(* IEC 61131-3 sources: Codesys/60-let-oktyabrya/src, 26 files *)

(* ---- E_PumpType.st ---- *)
(* ============================================================ *)
(* E_PumpType — тип преобразователя частоты ELHART             *)
(* ============================================================ *)
(* === ИЗМЕНЕНО === MINI удалён (в проектах его не было — была   *)
(* ошибка типа). Теперь два типа: PUMP (EMD-PUMP) и VL           *)
(* (EMD-VL/VH, векторный). Обработка обоих — в FB_Pump.          *)
(*                                                              *)
(* Тип каждого ПЧ задаётся в массиве GVL.ePumpType[1..cPumpCount] *)
(* (RETAIN). Автоопределение PUMP/VL по сигнатурному регистру —   *)
(* см. комментарий в PRG_Pumps (пока задаётся вручную).          *)
(* ============================================================ *)
TYPE E_PumpType :
(
    PUMP := 0,   // EMD-PUMP (F-коды, задание частоты в Гц ×100 → 0x2001)
    VL   := 1    // EMD-VL (P-группы, задание в % → 0x1000, статус 0x3000)
);
END_TYPE

(* ---- GVL.st ---- *)
(* ============================================================ *)
(* GVL — Глобальные переменные проекта "60 Лет Октября"         *)
(* (на основе ДДЮТ / Fontan_V1 / Саки Пруд)                     *)
(*                                                              *)
(* ШИНА Modbus RTU / RS-485:                                   *)
(*   COM1 (Modbus_COM), 9600/8/N/1:                            *)
(*     Адрес 1  — МВ110-16Д   (16 дискретных входов DI1..DI12) *)
(*     Адрес 2  — МУ110-16Р   (16 дискретных выходов DO1..DO4  *)
(*                используются, остальные свободны)             *)
(*   COM2 (Modbus_COM_2):                                       *)
(*     Адрес 41 — ELHART EMD-PUMP 1 (насос-шоу, индекс 1)      *)
(*     Адрес 42 — ELHART EMD-PUMP 2 (насос-шоу, индекс 2)      *)
(*     Адрес 43 — ELHART EMD-PUMP 3 (насос-шоу, индекс 3, НОВЫЙ)*)
(*     === 60ЛО:ВАЖНО === Устройство EMD_PUMP_3 нужно добавить  *)
(*     в дереве Modbus проекта (по аналогии с EMD_PUMP_1/2) —    *)
(*     без него PRG_Pumps.st (блок 4а) не скомпилируется.        *)
(*   ПЧ COM2 — насосы-шоу (не фильтрационные), просто            *)
(*   информационные, ни на что в логике не влияют.               *)
(* ============================================================ *)

(* ============================================================ *)
(* КОНСТАНТЫ СИСТЕМЫ                                            *)
(* ============================================================ *)
VAR_GLOBAL CONSTANT
    cPumpCount   : INT  := 3;        // === 60ЛО:ИЗМЕНЕНО === было 2 (ДДЮТ), теперь 3 насоса ПЧ (ПЧ1/ПЧ2/ПЧ3)
    cDI_Count    : INT  := 16;       // дискретных входов МВ110
    cDO_Count    : INT  := 16;       // дискретных выходов МУ110
    cMaxFreq     : REAL := 50.0;     // максимальная частота, Гц
    cMinFreq     : REAL := 0.0;      // минимальная частота, Гц
    cMinTime     : REAL := 0.1;      // мин. время разгона/торможения, с
    cMaxTime     : REAL := 6000.0;   // макс. время разгона/торможения, с
    cMaxCurrent  : REAL := 999.9;    // потолок номинального тока, А
    cMaxVoltage  : REAL := 500.0;    // потолок номинального напряжения, В
    cMaxOverheat : INT  := 150;      // потолок уровня перегрева, °C
    cMinOverheat : INT  := 40;       // минимум уровня перегрева, °C
END_VAR

(* ============================================================ *)
(* RETAIN-переменные (хранятся при отключении питания)         *)
(* ============================================================ *)
VAR_GLOBAL RETAIN
    (* Тип каждого ПЧ. Все три насоса — EMD-PUMP.                *)
    (* ВНИМАНИЕ: изменение требует Reset cold контроллера.      *)
    ePumpType : ARRAY[1..cPumpCount] OF E_PumpType :=
        [E_PumpType.PUMP, E_PumpType.PUMP, E_PumpType.PUMP];   // === 60ЛО:ИЗМЕНЕНО === добавлен 3-й элемент

    (* === ЖУРНАЛ ПЧ — БЕЗ ИЗМЕНЕНИЙ АРХИТЕКТУРЫ === *)
    (* Та же схема сдвига, что у журнала фонтана (см. подробный комментарий  *)
    (* в GVL_Fountain.st) — позиция 1 всегда самая свежая запись, при новой  *)
    (* записи всё сдвигается на 1 вниз, самая старая (позиция 30) выпадает.  *)
    (* Размер: 30 записей, длина ячейки 65.                                  *)
    (* ⚠️ С полными названиями возможна обрезка длинных строк — если         *)
    (* увидишь обрыв текста, увеличь до 80-90).                              *)
    aPumpLog       : ARRAY[1..30] OF WSTRING(65);
    iPumpLogCount  : INT;   // сколько записей реально заполнено (0..30)

    (* Флаг "задержка ошибки 0x02C0 уже записана в ПЧ" — RETAIN *)
    xErrDelayWritten : ARRAY[1..cPumpCount] OF BOOL := [cPumpCount(FALSE)];

    (* Флаг "параметр дисплея Fout (регистр 0) уже записан" — RETAIN *)
    xDispParamWritten : ARRAY[1..cPumpCount] OF BOOL := [cPumpCount(FALSE)];
END_VAR

(* ============================================================ *)
(* ГЛОБАЛЬНЫЕ ПЕРЕМЕННЫЕ                                        *)
(* ============================================================ *)
VAR_GLOBAL

    (* ========================================================= *)
    (* БЛОК 1: СОСТОЯНИЕ СИСТЕМЫ                                 *)
    (* ========================================================= *)
    xSystemState     : BOOL := TRUE;
    sSystemStateText : WSTRING(20);
    iErrors          : INT  := 0;
    iWorkCount       : INT  := 0;
    iStopCount       : INT  := 0;
    xAnyAlarm        : BOOL := FALSE;
    iErrorsPumps     : INT  := 0;
    iErrorsModules   : INT  := 0;
    iErrorsFountain  : INT  := 0;

    (* ========================================================= *)
    (* БЛОК 2: НАВИГАЦИЯ И ИНТЕРФЕЙС HMI                         *)
    (* ========================================================= *)
    xMenuOpen      : BOOL := TRUE;
    iCurrentScreen : INT  := 1;
    iSelPump       : INT  := 1;

    (* ========================================================= *)
    (* БЛОК 3: РЕЖИМ ОТЛАДКИ RS-485                              *)
    (* ========================================================= *)
    xDebugModeAll      : BOOL := FALSE;
    xDebugModeAll_Prev : BOOL := FALSE;

    xDebugModePump      : ARRAY[1..cPumpCount] OF BOOL := [cPumpCount(FALSE)];
    xDebugModePump_Prev : ARRAY[1..cPumpCount] OF BOOL := [cPumpCount(FALSE)];

    xApplyParamsAll  : BOOL := FALSE;
    xApplyParamsPump : ARRAY[1..cPumpCount] OF BOOL := [cPumpCount(FALSE)];

    (* ========================================================= *)
    (* ТРИГГЕРЫ ЧТЕНИЯ/ЗАПИСИ (конфигуратор-стиль)               *)
    (* ========================================================= *)
    xReadAllPump  : ARRAY[1..cPumpCount] OF BOOL := [cPumpCount(FALSE)];
    xReadAllAsk   : BOOL := FALSE;

    xWriteAllPump : ARRAY[1..cPumpCount] OF BOOL := [cPumpCount(FALSE)];
    xWriteAllAsk  : BOOL := FALSE;
    xWriteAllConfirm : BOOL := FALSE;

    xWr_AccTime      : ARRAY[1..cPumpCount] OF BOOL := [cPumpCount(FALSE)]; // 0x006B
    xWr_DecTime      : ARRAY[1..cPumpCount] OF BOOL := [cPumpCount(FALSE)]; // 0x006C
    xWr_MaxFreq      : ARRAY[1..cPumpCount] OF BOOL := [cPumpCount(FALSE)]; // 0x0069
    xWr_MinFreq      : ARRAY[1..cPumpCount] OF BOOL := [cPumpCount(FALSE)]; // 0x006A
    xWr_MotorCurrent : ARRAY[1..cPumpCount] OF BOOL := [cPumpCount(FALSE)]; // 0x00D2
    xWr_MotorVoltage : ARRAY[1..cPumpCount] OF BOOL := [cPumpCount(FALSE)]; // 0x00D1
    xWr_OverCurLevel : ARRAY[1..cPumpCount] OF BOOL := [cPumpCount(FALSE)]; // 0x01A7
    xWr_OverCurTime  : ARRAY[1..cPumpCount] OF BOOL := [cPumpCount(FALSE)]; // 0x01A8
    xWr_OverVoltProt : ARRAY[1..cPumpCount] OF BOOL := [cPumpCount(FALSE)]; // 0x019B
    xWr_Overheat     : ARRAY[1..cPumpCount] OF BOOL := [cPumpCount(FALSE)]; // 0x0325
    xWr_OverCurAcc   : ARRAY[1..cPumpCount] OF BOOL := [cPumpCount(FALSE)]; // 0x0199

    xWr_UnlockF800   : ARRAY[1..cPumpCount] OF BOOL := [cPumpCount(FALSE)]; // 0x0320
    xWr_Sources      : ARRAY[1..cPumpCount] OF BOOL := [cPumpCount(FALSE)]; // 0x0065/0x0066

    xWritePending    : ARRAY[1..cPumpCount] OF BOOL := [cPumpCount(FALSE)];
    xWaitStopForWrite : ARRAY[1..cPumpCount] OF BOOL := [cPumpCount(FALSE)];

    (* === 60ЛО:УДАЛИТЬ ===                                       *)
    (* Раньше использовался для запроса физической остановки      *)
    (* фильтр.насоса через лампы DO6/DO8 перед записью параметров. *)
    (* Не читается нигде физически, оставлен только для истории.  *)
    xReqStopFiltrForWrite : ARRAY[1..cPumpCount] OF BOOL := [cPumpCount(FALSE)];

    xFactoryResetAll  : BOOL := FALSE;
    xFactoryResetPump : ARRAY[1..cPumpCount] OF BOOL := [cPumpCount(FALSE)];

    wCmdSourceWrite  : ARRAY[1..cPumpCount] OF WORD := [cPumpCount(WORD#1)];
    wFreqSourceWrite : ARRAY[1..cPumpCount] OF WORD := [cPumpCount(WORD#3)];

    (* ========================================================= *)
    (* БЛОК 4: МВ110-16Д — ДИСКРЕТНЫЕ ВХОДЫ                      *)
    (* ========================================================= *)
    wMV110_Inputs : WORD;
    xMV110_Error  : BOOL;
    xDI           : ARRAY[1..cDI_Count] OF BOOL;
    (* Используются DI1..DI12. Карта DI — см. PRG_Fountain блок 2. *)

    (* ========================================================= *)
    (* БЛОК 5: МУ110-16Р — ДИСКРЕТНЫЕ ВЫХОДЫ                     *)
    (* ========================================================= *)
    (* === 60ЛО:ИЗМЕНЕНО === Карта DO1..DO4 — см. PRG_Fountain     *)
    (* блок 15. DO1 сухой ход (дубляж DI4), DO2 насосы фонтана,    *)
    (* DO3 подсветка, DO4 клапан добора (дубляж DI5). Остальные    *)
    (* DO свободны.                                                *)
    xDO                : ARRAY[1..cDO_Count] OF BOOL := [cDO_Count(FALSE)];

    wMU110_Outputs     : WORD := 0;
    wMU110_OutputsRead : WORD;
    xMU110_Error       : BOOL;

    wMU110_SafeOutputs : WORD := 0;
    xMU110_WriteSafe   : BOOL := FALSE;

    (* ========================================================= *)
    (* БЛОК 6: НАСОСЫ — ЭКЗЕМПЛЯРЫ ФУНКЦИОНАЛЬНЫХ БЛОКОВ         *)
    (* ========================================================= *)
    Pump : ARRAY[1..cPumpCount] OF FB_Pump;

    (* ========================================================= *)
    (* БЛОК 7: НАСОСЫ — ЗАДАНИЕ ОПЕРАТОРА (_Set)                 *)
    (* ========================================================= *)
    xPumpRunCmd : ARRAY[1..cPumpCount] OF BOOL := [cPumpCount(FALSE)];

    rPumpFreqSetHz          : ARRAY[1..cPumpCount] OF REAL := [cPumpCount(40.0)];
    rPumpAccTime_Set        : ARRAY[1..cPumpCount] OF REAL := [10.0, 10.0, 10.0];   // === 60ЛО:ИЗМЕНЕНО === было [10.0, 10.0]
    rPumpDecTime_Set        : ARRAY[1..cPumpCount] OF REAL := [10.0, 10.0, 10.0];   // === 60ЛО:ИЗМЕНЕНО === было [10.0, 10.0]
    rPumpMaxFreq_Set        : ARRAY[1..cPumpCount] OF REAL := [cPumpCount(40.0)];
    rPumpMinFreq_Set        : ARRAY[1..cPumpCount] OF REAL := [cPumpCount(0.0)];
    rPumpMotorRatedCurrent_Set : ARRAY[1..cPumpCount] OF REAL := [cPumpCount(14.9)];
    rPumpMotorRatedVoltage_Set : ARRAY[1..cPumpCount] OF REAL := [cPumpCount(380.0)];
    rPumpOverCurrentLevel_A_Set : ARRAY[1..cPumpCount] OF REAL := [cPumpCount(26.1)];
    rPumpOverCurrentTime_Set    : ARRAY[1..cPumpCount] OF REAL := [cPumpCount(5.0)];
    xPumpOverVoltProtect_Set    : ARRAY[1..cPumpCount] OF BOOL := [cPumpCount(TRUE)];
    iPumpOverheatLevel_Set      : ARRAY[1..cPumpCount] OF INT  := [cPumpCount(95)];
    iPumpOverCurAcc_Set         : ARRAY[1..cPumpCount] OF INT  := [cPumpCount(150)];

    (* ========================================================= *)
    (* БЛОК 7а: ОТЛАДКА — групповые команды и флаги окон        *)
    (* ========================================================= *)
    xDbgRunAll  : BOOL;
    xDbgStopAll : BOOL;

    xAskApply   : BOOL := FALSE;
    xAskFactory : BOOL := FALSE;
	xAskDialogStopPch : BOOL := FALSE;

    (* ========================================================= *)
    (* БЛОК 8: НАСОСЫ — ДАННЫЕ ДЛЯ ОТОБРАЖЕНИЯ НА HMI            *)
    (* ========================================================= *)
    xPumpWork      : ARRAY[1..cPumpCount] OF BOOL;
    xPumpStop      : ARRAY[1..cPumpCount] OF BOOL;
    xPumpAlarm     : ARRAY[1..cPumpCount] OF BOOL;
    xPumpReverse   : ARRAY[1..cPumpCount] OF BOOL;
    xPumpCommError : ARRAY[1..cPumpCount] OF BOOL;
    xPumpCommRaw   : ARRAY[1..cPumpCount] OF BOOL;
    tonPumpCommFilter : ARRAY[1..cPumpCount] OF TON;

    sPumpState         : ARRAY[1..cPumpCount] OF WSTRING(50);
    sPumpFaultText      : ARRAY[1..cPumpCount] OF WSTRING(100);
    sPumpTypeText       : ARRAY[1..cPumpCount] OF WSTRING(20);
    sPumpFaultLastText  : ARRAY[1..cPumpCount] OF WSTRING(100);
    sPumpFault2Text     : ARRAY[1..cPumpCount] OF WSTRING(100);
    sPumpFault3Text     : ARRAY[1..cPumpCount] OF WSTRING(100);
    sPumpFault4Text     : ARRAY[1..cPumpCount] OF WSTRING(100);

    rPumpFreqSetActHz : ARRAY[1..cPumpCount] OF REAL;
    rPumpFreqActHz    : ARRAY[1..cPumpCount] OF REAL;
    rPumpCurrentActA  : ARRAY[1..cPumpCount] OF REAL;
    rPumpSpeedActRpm  : ARRAY[1..cPumpCount] OF REAL;
    rPumpDcVoltageV   : ARRAY[1..cPumpCount] OF REAL;
    iPumpTemperatureC : ARRAY[1..cPumpCount] OF INT;
    rPumpVoltageActV  : ARRAY[1..cPumpCount] OF REAL;
    rPumpRuntimeHours : ARRAY[1..cPumpCount] OF REAL;

    dwPumpLampColor : ARRAY[1..cPumpCount] OF DWORD;

    rPumpAccTime_Disp            : ARRAY[1..cPumpCount] OF REAL;
    rPumpDecTime_Disp            : ARRAY[1..cPumpCount] OF REAL;
    rPumpMaxFreq_Disp            : ARRAY[1..cPumpCount] OF REAL;
    rPumpMinFreq_Disp            : ARRAY[1..cPumpCount] OF REAL;
    rPumpMotorRatedCurrent_Disp  : ARRAY[1..cPumpCount] OF REAL;
    rPumpMotorRatedVoltage_Disp  : ARRAY[1..cPumpCount] OF REAL;
    rPumpOverCurrentLevel_A_Disp : ARRAY[1..cPumpCount] OF REAL;
    rPumpOverCurrentTime_Disp    : ARRAY[1..cPumpCount] OF REAL;
    xPumpOverVoltProtect_Disp    : ARRAY[1..cPumpCount] OF BOOL;
    sPumpOverVoltProtect : ARRAY[1..cPumpCount] OF WSTRING(20);
    iPumpOverCurrentLevel_pct_Disp : ARRAY[1..cPumpCount] OF INT;
    iPumpOverheatLevel_Disp      : ARRAY[1..cPumpCount] OF INT;
    iPumpOverCurAcc_Disp         : ARRAY[1..cPumpCount] OF INT;

    (* ========================================================= *)
    (* БЛОК 9: НАСОСЫ — ЗАПИСЬ В ПЧ (Modbus WRITE)               *)
    (* ========================================================= *)
    wPumpCmd  : ARRAY[1..cPumpCount] OF WORD;
    wPumpFreq : ARRAY[1..cPumpCount] OF WORD;

    wPumpAccTimeWrite           : ARRAY[1..cPumpCount] OF WORD;
    wPumpDecTimeWrite           : ARRAY[1..cPumpCount] OF WORD;
    wPumpMaxFreqWrite           : ARRAY[1..cPumpCount] OF WORD;
    wPumpMinFreqWrite           : ARRAY[1..cPumpCount] OF WORD;
    wPumpMotorRatedCurrentWrite : ARRAY[1..cPumpCount] OF WORD;
    wPumpMotorRatedVoltageWrite : ARRAY[1..cPumpCount] OF WORD;
    wPumpOverCurrentLevelWrite  : ARRAY[1..cPumpCount] OF WORD;
    wPumpOverCurrentTimeWrite   : ARRAY[1..cPumpCount] OF WORD;
    wPumpOverVoltProtectWrite   : ARRAY[1..cPumpCount] OF WORD;
    wPumpOverheatLevelWrite     : ARRAY[1..cPumpCount] OF WORD;
    wPumpOverCurAccWrite        : ARRAY[1..cPumpCount] OF WORD;

    wPumpDispParamWrite : ARRAY[1..cPumpCount] OF WORD := [cPumpCount(WORD#1)];

    wPumpRS_ErrDelayWrite : ARRAY[1..cPumpCount] OF WORD := [cPumpCount(WORD#5)];
    xWr_ErrDelayInit      : ARRAY[1..cPumpCount] OF BOOL := [cPumpCount(FALSE)];

    wPumpExtSettingsUnlockWrite : ARRAY[1..cPumpCount] OF WORD;
    wPumpFactoryResetWrite      : ARRAY[1..cPumpCount] OF WORD := [cPumpCount(WORD#0)];

    (* ========================================================= *)
    (* БЛОК 10: НАСОСЫ — ЧТЕНИЕ ИЗ ПЧ (Modbus READ)             *)
    (* ========================================================= *)
    wPumpFreqSetRead     : ARRAY[1..cPumpCount] OF WORD;
    wPumpFreqActual      : ARRAY[1..cPumpCount] OF WORD;
    wPumpCurrentActual   : ARRAY[1..cPumpCount] OF WORD;
    wPumpSpeedActual     : ARRAY[1..cPumpCount] OF WORD;
    wPumpDcVoltage       : ARRAY[1..cPumpCount] OF WORD;
    wPumpTemperature     : ARRAY[1..cPumpCount] OF WORD;
    wPumpPidFeedback     : ARRAY[1..cPumpCount] OF WORD;
    wPumpRuntimeHoursRaw : ARRAY[1..cPumpCount] OF WORD;
    wPumpVoltageActual   : ARRAY[1..cPumpCount] OF WORD;

    wPumpFaultLast : ARRAY[1..cPumpCount] OF WORD;
    wPumpFault2    : ARRAY[1..cPumpCount] OF WORD;
    wPumpFault3    : ARRAY[1..cPumpCount] OF WORD;
    wPumpFault4    : ARRAY[1..cPumpCount] OF WORD;

    wPumpFaultReg : ARRAY[1..cPumpCount] OF WORD;
    wPumpStatus   : ARRAY[1..cPumpCount] OF WORD;
    wPumpStopState    : ARRAY[1..cPumpCount] OF WORD;
    xPumpFullyStopped : ARRAY[1..cPumpCount] OF BOOL;

    wPumpFreqPresetRead  : ARRAY[1..cPumpCount] OF WORD;
    rPumpFreqPresetHz : ARRAY[1..cPumpCount] OF REAL;
    wPumpFreqSourceRead  : ARRAY[1..cPumpCount] OF WORD;
    wPumpCmdSourceRead   : ARRAY[1..cPumpCount] OF WORD;
    wPumpStopKeyLockRead : ARRAY[1..cPumpCount] OF WORD;
    wPumpReverseLockRead : ARRAY[1..cPumpCount] OF WORD;
    wPumpMaxFreqRead     : ARRAY[1..cPumpCount] OF WORD;
    wPumpMinFreqRead     : ARRAY[1..cPumpCount] OF WORD;
    wPumpAccTimeRaw      : ARRAY[1..cPumpCount] OF WORD;
    wPumpDecTimeRaw      : ARRAY[1..cPumpCount] OF WORD;

    wPumpStartMethodRead        : ARRAY[1..cPumpCount] OF WORD;
    wPumpStopMethodRead         : ARRAY[1..cPumpCount] OF WORD;
    wPumpStartFreqRead          : ARRAY[1..cPumpCount] OF WORD;
    wPumpStopFreqRead           : ARRAY[1..cPumpCount] OF WORD;
    wPumpMotorRatedVoltageRead  : ARRAY[1..cPumpCount] OF WORD;
    wPumpMotorRatedCurrentRead  : ARRAY[1..cPumpCount] OF WORD;
    wPumpMotorNoLoadCurrentRead : ARRAY[1..cPumpCount] OF WORD;
    wPumpMotorRatedSpeedRead    : ARRAY[1..cPumpCount] OF WORD;

    wPumpFIV_MinRead    : ARRAY[1..cPumpCount] OF WORD;
    wPumpFIV_MaxRead    : ARRAY[1..cPumpCount] OF WORD;
    wPumpFIV_FilterRead : ARRAY[1..cPumpCount] OF WORD;
    wPumpFIC_MinRead    : ARRAY[1..cPumpCount] OF WORD;
    wPumpFIC_MaxRead    : ARRAY[1..cPumpCount] OF WORD;

    wPumpFOV_MinRead : ARRAY[1..cPumpCount] OF WORD;
    wPumpFOV_MaxRead : ARRAY[1..cPumpCount] OF WORD;
    wPumpFOC_MinRead : ARRAY[1..cPumpCount] OF WORD;
    wPumpFOC_MaxRead : ARRAY[1..cPumpCount] OF WORD;

    wPumpAI_MinFreqRead  : ARRAY[1..cPumpCount] OF WORD;
    wPumpAI_MinDirRead   : ARRAY[1..cPumpCount] OF WORD;
    wPumpAI_MaxFreqRead  : ARRAY[1..cPumpCount] OF WORD;
    wPumpAI_MaxDirRead   : ARRAY[1..cPumpCount] OF WORD;
    wPumpAI_ReverseEnRead: ARRAY[1..cPumpCount] OF WORD;

    wPumpDI_FWD_Read : ARRAY[1..cPumpCount] OF WORD;
    wPumpDI_REV_Read : ARRAY[1..cPumpCount] OF WORD;
    wPumpDI_S1_Read  : ARRAY[1..cPumpCount] OF WORD;
    wPumpDI_S2_Read  : ARRAY[1..cPumpCount] OF WORD;
    wPumpDI_S3_Read  : ARRAY[1..cPumpCount] OF WORD;
    wPumpDI_S4_Read  : ARRAY[1..cPumpCount] OF WORD;
    wPumpDI_S5_Read  : ARRAY[1..cPumpCount] OF WORD;
    wPumpDI_S6_Read  : ARRAY[1..cPumpCount] OF WORD;

    wPumpDO_M01_Read   : ARRAY[1..cPumpCount] OF WORD;
    wPumpDO_M02_Read   : ARRAY[1..cPumpCount] OF WORD;
    wPumpDO_Relay_Read : ARRAY[1..cPumpCount] OF WORD;

    wPumpOverCurAccRead       : ARRAY[1..cPumpCount] OF WORD;
    wPumpOverCurSteadyRead    : ARRAY[1..cPumpCount] OF WORD;
    wPumpOverVoltProtectRead  : ARRAY[1..cPumpCount] OF WORD;
    wPumpOverCurReactionRead  : ARRAY[1..cPumpCount] OF WORD;
    wPumpOverCurrentLevelRead : ARRAY[1..cPumpCount] OF WORD;
    wPumpOverCurrentTimeRead  : ARRAY[1..cPumpCount] OF WORD;
    wPumpOverheatLevelRead    : ARRAY[1..cPumpCount] OF WORD;

    wPumpRS_BaudRead      : ARRAY[1..cPumpCount] OF WORD;
    wPumpRS_FormatRead    : ARRAY[1..cPumpCount] OF WORD;
    wPumpRS_AddrRead      : ARRAY[1..cPumpCount] OF WORD;
    wPumpRS_ErrActionRead : ARRAY[1..cPumpCount] OF WORD;
    wPumpRS_ErrDelayRead  : ARRAY[1..cPumpCount] OF WORD;

    (* ========================================================= *)
    (* БЛОК 11: VISU DEBUG — ВЫБОР НАСОСА И ДИАЛОГИ              *)
    (* ========================================================= *)
    (* === 60ЛО:ИЗМЕНЕНО === iDebugPumpSelected теперь может быть 1..3 *)
    iDebugMode         : INT;
    iDebugPumpSelected : INT := 1;
    xDlgConfirmApply   : BOOL;
    xDlgConfirmFactory : BOOL;

(* ========================================================= *)
(* БЛОК 12: ЖУРНАЛ ИЗМЕНЕНИЙ ПАРАМЕТРОВ ПЧ *)
(* ========================================================= *)
xLogClear : BOOL := FALSE;
xAskClearLog : BOOL := FALSE;

rLog_AccTime_Prev : ARRAY[1..cPumpCount] OF REAL;
rLog_DecTime_Prev : ARRAY[1..cPumpCount] OF REAL;
rLog_MaxFreq_Prev : ARRAY[1..cPumpCount] OF REAL;
rLog_MinFreq_Prev : ARRAY[1..cPumpCount] OF REAL;
rLog_MotorCur_Prev : ARRAY[1..cPumpCount] OF REAL;
rLog_MotorVolt_Prev : ARRAY[1..cPumpCount] OF REAL;
rLog_OCLevel_Prev : ARRAY[1..cPumpCount] OF REAL;
rLog_OCTime_Prev : ARRAY[1..cPumpCount] OF REAL;
xLog_OVProt_Prev : ARRAY[1..cPumpCount] OF BOOL;
iLog_Overheat_Prev : ARRAY[1..cPumpCount] OF INT;
iLog_OCAcc_Prev : ARRAY[1..cPumpCount] OF INT;
xLog_Initialized : ARRAY[1..cPumpCount] OF BOOL := [cPumpCount(FALSE)];
rtrigReadAll_Prev : ARRAY[1..cPumpCount] OF BOOL := [cPumpCount(FALSE)];

xWr_DispParam : ARRAY[1..cPumpCount] OF BOOL := [cPumpCount(FALSE)];
END_VAR

(* ---- GVL_Fountain.st ---- *)
(* ============================================================ *)
(* GVL_Fountain — переменные автоматики "60 Лет Октября"        *)
(* (на основе ДДЮТ / Саки Пруд)                                 *)
(*                                                              *)
(* === 60ЛО: ГЛАВНЫЕ ОТЛИЧИЯ ОТ ДДЮТ ===                        *)
(*  - Дозация (pH/альгицид/биопаг) на другом контроллере.       *)
(*  - Добор воды решает Мусидора — мы зеркалим DI5→DO4,         *)
(*    проверяем DI6 (20с).                                      *)
(*  - Только 4 физических DO. У света/насосов появилось         *)
(*    подтверждение реле (DI9/DI10, 2с).                        *)
(*  - ПР200 и резерв полива СПК не нужны вообще.                *)
(*                                                              *)
(* ВАЖНО: переменные, оставшиеся от ДДЮТ и не задействованные   *)
(* в новой логике, НЕ УДАЛЕНЫ — только помечены комментарием    *)
(* "60ЛО: не используется" — их значение ничем не пишется, но   *)
(* они остаются объявленными, чтобы не ломать привязки экранов. *)
(* Финальное решение по удалению — за тобой после проверки.     *)
(* ============================================================ *)

VAR_GLOBAL CONSTANT
    (* === ДДЮТ:УДАЛИТЬ — шкала уровня чаши по AI1, не нужна === *)
    (*
    cWaterRawMin : REAL := 4.0;
    cWaterRawMax : REAL := 20.0;
    cWaterCmMin  : REAL := 0.0;
    cWaterCmMax  : REAL := 100.0;
    *)

    (* 60ЛО: не используется — были нужны только для *)
    (* PRG_PolivSPK.st, который выводится из проекта. *)
    cSlivRawMin : REAL := 4.0;
    cSlivRawMax : REAL := 20.0;
    cSlivCmMin  : REAL := 0.0;
    cSlivCmMax  : REAL := 100.0;
END_VAR

VAR_GLOBAL RETAIN
    aFountainLog       : ARRAY[1..60] OF WSTRING(60);
    iFountainLogCount  : INT;

    iAdminPassCorrect : INT := 1234;

    (* ===== ГЛАВНЫЕ ТУМБЛЕРЫ С ЭКРАНА ====================== *)
    xVseSist : BOOL := TRUE;
    iPumpSelect : INT := 2;   // насосы фонтана: 0=ручной,1=выкл,2=авто

    xNfEnable : BOOL := TRUE;   // 60ЛО: не используется в новой логике (была тупиковой ещё в ДДЮТ), оставлено для визуализации

    (* 60ЛО: не используется — старая система 2/3 датчиков и гистерезисов уровня. *)
    (* Добор полностью решает Мусидора, мы клапаном не управляем.                 *)
    iLevelSensorCountPending : INT := 2;
    tLevel1DebounceSec : INT := 20;
    tLevel2DebounceSec : INT := 20;
    tLevel3DebounceSec : INT := 20;
    iRefillOffDelayMin : INT := 2;
    iRefillOffDelaySec : INT := 0;

    iTimeZoneOffsetSec : INT := 10800;   // смещение часового пояса от UTC, сек

    iUvNfMinRunMin : INT := 20;   // 60ЛО: не используется (выхода на УФ нет, был информационным и в ДДЮТ)

    (* 60ЛО: не используется — старая система попыток добора. *)
    tRefillDurHours     : INT := 2;
    tBetweenRefillHours : INT := 12;
    iRefillAttemptsMax  : INT := 5;

    (* 60ЛО: не используется — дозация на другом контроллере. Экраны pH/альгицид/биопаг скрыты из меню. *)
    iPhSelect : INT := 2;
    iAlgSelect        : INT := 2;
    rAlgDoseMlPerDay  : REAL := 66.0;
    rAlgFlowMlPerHour : REAL := 1125.0;
    iBioSelect        : INT := 2;
    rBioDoseMlPerDay  : REAL := 33.0;
    rBioFlowMlPerHour : REAL := 1154.0;

    (* ===== ОКНО ИСПРАВНОСТИ ФИЛЬТРАЦИИ — АКТИВНО, счётчик промывок сохранён === *)
    iFilterMinRunMin   : INT := 30;    // порог наработки НФ, мин
    iFilterWindowHours : INT := 12;    // 60ЛО: не используется (устар. ещё в ДДЮТ)
    iNfHealthyWindowMin : INT := 0;    // 60ЛО: не используется (устар. ещё в ДДЮТ)

    (* === СЧЁТЧИК ПРОМЫВОК НФ — АКТИВНО, БЕЗ ИЗМЕНЕНИЙ АЛГОРИТМА === *)
    iNfLastOnHour  : INT;
    iNfLastOnMin   : INT;
    iNfLastOnDay   : INT;
    iNfLastOnMonth : INT;
    iNfLastOnYear  : INT;
    iNfFlushStage  : INT;
    xNfFlushReady  : BOOL := TRUE;
    iNfFlushCount  : INT;
    iNfFlushHour   : INT;
    iNfFlushMin    : INT;
    iNfFlushDay    : INT;
    iNfFlushMonth  : INT;
    iNfFlushYear   : INT;

    iNfRunMinAccum    : INT;    // 60ЛО: не используется (устар. ещё в ДДЮТ)
    iNfRunSecAccum    : DINT;   // 60ЛО: не используется (устар. ещё в ДДЮТ)
    iNfHealthySecLeft : DINT;   // 60ЛО: не используется (устар. ещё в ДДЮТ)
    iNfHealthyHoursLeft : INT;  // 60ЛО: не используется (устар. ещё в ДДЮТ)
    iNfHealthyMinLeft   : INT;  // 60ЛО: не используется (устар. ещё в ДДЮТ)
    xNfProven         : BOOL;   // 60ЛО: не используется (устар. ещё в ДДЮТ)
    xNfWorkPrev       : BOOL;   // АКТИВНО — детект фронта для счётчика промывок
    iNfContinuousRunHour : INT;
    iNfContinuousRunMin  : INT;
    iNfContinuousRunSec  : INT;

    xNfFirstScanDone : BOOL;
    iNfJustEndedSec  : INT;

    xZapretDozacii : BOOL := TRUE;   // 60ЛО: не используется (дозация на другом контроллере)

    iDamperSelect : INT := 2;   // 60ЛО: не используется — заслонка теперь просто зеркало DI5→DO4

    (* ===== СВЕТ — АКТИВНО ==================================== *)
    iLightSelect : INT  := 2;       // свет: 0=ручной,1=выкл,2=авто(закат)
    iSoundMode   : INT  := 2;       // FUTURE_SOUND, не используется
    xSoundEnable : BOOL := TRUE;    // FUTURE_SOUND, не используется

    (* ===== РАСЧЁТ ЗАКАТА — АКТИВНО, БЕЗ ИЗМЕНЕНИЙ ============== *)
    rSunLatitude          : REAL := 44.61581;
    rSunLongitude         : REAL := 33.52276;
    rSunLongitudePrev     : REAL := 33.52276;
    iChoseTimeZone        : INT  := 14;
    iSunsetCorrectSigned  : INT  := 0;

    iOffHourWeekday    : INT := 23;
    iOffMinuteWeekday  : INT := 0;
    iOffHourWeekend    : INT := 23;
    iOffMinuteWeekend  : INT := 0;

    iLightScheduleMode : INT := 3;   // 0=Авто,1=Вкл,2=Выкл,3=Астро
    iPumpScheduleMode  : INT := 0;   // 0=Авто,1=Вкл,2=Выкл

    iLightOnHourWeekday   : INT := 18;
    iLightOnMinuteWeekday : INT := 0;
    iLightOnHourWeekend   : INT := 18;
    iLightOnMinuteWeekend : INT := 0;

    iPumpOnHourWeekday    : INT := 8;
    iPumpOnMinuteWeekday  : INT := 0;
    iPumpOnHourWeekend    : INT := 8;
    iPumpOnMinuteWeekend  : INT := 0;

    (* 60ЛО: не используется — накопители ручной наработки НФ/pH из ДДЮТ. *)
    iNfManualRunMinBuffer : INT;
    iNfManualRunMinToday  : INT;
    iNfManualRunHourTotal : INT;
    iPhManualRunMinBuffer : INT;
    iAlgManualRunMinBuffer : INT;
    iPhManualRunSecAccum : DINT;
    iPhManRunSec  : INT;
    iPhManRunHour : INT;
    iPhManRunMin  : INT;

    (* 60ЛО: не используется — накопленная наработка дозаторов, дозация не наша. *)
    iPhRunHourTotal : INT;
    iAlgRunHour : INT;
    iAlgRunMinBuffer2 : INT;
    iPhRunSecAccum : DINT;
    iPhRunSecDisp  : INT;
    iAlgRunSecAccum : DINT;
    iAlgRunSec  : INT;
    iPhStartCount  : INT;
    iAlgStartCount  : INT;

    (* 60ЛО: не используется — долговая система альгицида/биопага. *)
    rAlgDebtSec         : REAL := 0.0;
    udiAlgLastDebtStamp : UDINT := 0;
    xAlgDebtInitDone    : BOOL := FALSE;
    iAlgLastDoseDay     : INT := 0;
    iAlgLastDoseMonth   : INT := 0;
    iAlgLastDoseYear    : INT := 0;
    iAlgLastDoseHourR   : INT := 0;
    iAlgLastDoseMinR    : INT := 0;
    iAlgLastDoseSecR    : INT := 0;

    rBioDebtSec         : REAL := 0.0;
    udiBioLastDebtStamp : UDINT := 0;
    xBioDebtInitDone    : BOOL := FALSE;
    iBioLastDoseDay     : INT := 0;
    iBioLastDoseMonth   : INT := 0;
    iBioLastDoseYear    : INT := 0;
    iBioLastDoseHourR   : INT := 0;
    iBioLastDoseMinR    : INT := 0;
    iBioLastDoseSecR    : INT := 0;
    iBioRunSecAccum     : DINT;
    iBioRunSecDisp      : INT;
    iBioStartCount      : INT;
    iBioManSetMin    : INT := 10;
    iBioManRemMinRaw    : INT;
    iBioManRemSecRaw    : INT;
END_VAR

VAR_GLOBAL
    (* ===== ЖУРНАЛ ИЗМЕНЕНИЙ ФОНТАНА — АКТИВНО, БЕЗ ИЗМЕНЕНИЙ === *)
    xAskClearFountainLog     : BOOL;
    iFountainLogPinEntry     : INT;
    xFountainLogPinSubmit    : BOOL;
    xFountainLogClearedMsg   : BOOL;
    xFountainLogPassBadMsg   : BOOL;
    xFountainLogClear        : BOOL;

    iPumpLogPinEntry     : INT;
    xPumpLogPinSubmit    : BOOL;
    xPumpLogClearedMsg   : BOOL;
    xPumpLogPassBadMsg   : BOOL;

    xFountainLogInitialized : BOOL;

    (* "Тени" отслеживаемых параметров — те, что реально сравниваются в новой *)
    (* логике, помечены АКТИВНО, остальные (были в ДДЮТ) — не используются.  *)
    iLogPrevFilterMinRunMin  : INT;   // АКТИВНО
    iLogPrevUvNfMinRunMin    : INT;   // 60ЛО: не используется
    rLogPrevAlgDoseMlPerDay  : REAL;  // 60ЛО: не используется
    rLogPrevAlgFlowMlPerHour : REAL;  // 60ЛО: не используется
    rLogPrevBioDoseMlPerDay  : REAL;  // 60ЛО: не используется
    rLogPrevBioFlowMlPerHour : REAL;  // 60ЛО: не используется
    iLogPrevAlgManSetMin     : INT;   // 60ЛО: не используется
    iLogPrevBioManSetMin     : INT;   // 60ЛО: не используется
    iLogPrevPhSelect         : INT;   // 60ЛО: не используется
    iLogPrevAlgSelect        : INT;   // 60ЛО: не используется
    iLogPrevBioSelect        : INT;   // 60ЛО: не используется
    xLogPrevVseSist          : BOOL;  // АКТИВНО
    iLogPrevDamperSelect     : INT;   // 60ЛО: не используется
    iLogPrevLightSelect      : INT;   // АКТИВНО
    iLogPrevPumpSelect       : INT;   // АКТИВНО
    iLogPrevLevelSensorCount : INT;   // 60ЛО: не используется
    iLogPrevLightScheduleMode : INT;  // АКТИВНО
    iLogPrevPumpScheduleMode  : INT;  // АКТИВНО
    iLogPrevLightOnHourWeekday   : INT;   // АКТИВНО
    iLogPrevLightOnMinuteWeekday : INT;   // АКТИВНО
    iLogPrevLightOnHourWeekend   : INT;   // АКТИВНО
    iLogPrevLightOnMinuteWeekend : INT;   // АКТИВНО
    iLogPrevPumpOnHourWeekday    : INT;   // АКТИВНО
    iLogPrevPumpOnMinuteWeekday  : INT;   // АКТИВНО
    iLogPrevPumpOnHourWeekend    : INT;   // АКТИВНО
    iLogPrevPumpOnMinuteWeekend  : INT;   // АКТИВНО
    iLogPrevOffHourWeekday       : INT;   // АКТИВНО
    iLogPrevOffMinuteWeekday     : INT;   // АКТИВНО
    iLogPrevOffHourWeekend       : INT;   // АКТИВНО
    iLogPrevOffMinuteWeekend     : INT;   // АКТИВНО
    iLogPrevSunsetCorrectSigned  : INT;   // АКТИВНО
    iLogPrevChoseTimeZone        : INT;   // АКТИВНО
    rLogPrevSunLatitude          : REAL;  // АКТИВНО
    rLogPrevSunLongitude         : REAL;  // АКТИВНО
    xLogPrevAlarmReset       : BOOL;      // АКТИВНО
    iLogPrevLevel1DebounceSec   : INT;    // 60ЛО: не используется
    iLogPrevLevel2DebounceSec   : INT;    // 60ЛО: не используется
    iLogPrevLevel3DebounceSec   : INT;    // 60ЛО: не используется
    iLogPrevRefillOffDelayMin   : INT;    // 60ЛО: не используется
    iLogPrevRefillOffDelaySec   : INT;    // 60ЛО: не используется
    iLogPrevRefillDurHours      : INT;    // 60ЛО: не используется
    iLogPrevBetweenRefillHours  : INT;    // 60ЛО: не используется
    iLogPrevRefillAttemptsMax   : INT;    // 60ЛО: не используется

    rSlivRaw     : REAL;    // 60ЛО: не используется (был для PRG_PolivSPK.st)
    rSlivLevelCm : REAL;    // 60ЛО: не используется

    (* ===== СУХОЙ ХОД ============================================ *)
    xLevel1   : BOOL;   // 60ЛО: не используется — старая система 2/3 датчиков
    xLevel2   : BOOL;   // 60ЛО: не используется
    xLevel3   : BOOL;   // 60ЛО: не используется

    xPump1Work : BOOL;   // ← DI1, информационный
    xPump2Work : BOOL;   // ← DI2, информационный
    xPump3Work : BOOL;   // ← DI3, информационный, НОВЫЙ

    xDryRunOk    : BOOL;   // ← DI4, 1=норма (сигнал уже готов от Мусидоры)
    xDryRunAlarm : BOOL;   // = NOT xDryRunOk, ЖИВАЯ, САМАЯ ПЕРВАЯ авария в списке
    xDryRunRelayFb    : BOOL;   // ← DI8, подтверждение реле сухого хода
    xDryRunRelayAlarm : BOOL;   // авария: DO1 и DI8 разошлись >2с (защёлка)

    xLevel2LowConfirmed  : BOOL;  // 60ЛО: не используется
    xLevel2HighConfirmed : BOOL;  // 60ЛО: не используется
    xLevel3HighConfirmed : BOOL;  // 60ЛО: не используется
    xRefillStartConfirmed : BOOL; // 60ЛО: не используется
    xRefillEnoughConfirmed : BOOL; // 60ЛО: не используется
    xRefillOffConfirmed : BOOL;   // 60ЛО: не используется

    (* ===== КЛАПАН ДОБОРА — простое зеркало DI5→DO4 ============= *)
    xDamperCmdOpen    : BOOL;        // 60ЛО: не используется — старая логика управления клапаном
    xDamperCmdRaw     : BOOL;        // ← DI5, "пуск добора" от Мусидоры, копируется на DO4
    xDamperForceOpen   : BOOL;       // 60ЛО: не используется
    xDamperForceClose  : BOOL;       // 60ЛО: не используется
    xDamperZapretDobor : BOOL;       // 60ЛО: не используется
    xDamperRelayFb   : BOOL;         // ← DI6, подтверждение положения клапана
    xDamperRelayAlarm : BOOL;        // авария: DO4 и DI6 разошлись >20с (защёлка)
    sDamperPosition   : WSTRING(20); // "Открыт" / "Закрыт" (по DI6)
    sDamperFullStatus : WSTRING(50); // 60ЛО: не используется

    xOnlyTwoLevels : BOOL;   // 60ЛО: не используется
    iRefillAttempts   : INT;   // 60ЛО: не используется
    xRefillPauseRun   : BOOL;  // 60ЛО: не используется
    xRefillAttemptsAlarm : BOOL;  // 60ЛО: не используется

    (* ===== РАЗРЕШЕНИЯ И ФИЛЬТРАЦИЯ ======================= *)
    xPermissionToWork : BOOL;        // = xVseSist AND NOT xDryRunAlarm, общий статус для визуализации
    xNfWork           : BOOL;        // ← DI7, контактор фильтрации (НФ физически работает)
    xNfHealthy        : BOOL;        // непрерывная наработка НФ ≥ iFilterMinRunMin
    xNfPermission     : BOOL;        // 60ЛО: не используется
    xBlokDozacii      : BOOL;        // 60ЛО: не используется
    xFiltrationBlock  : BOOL;        // 60ЛО: не используется (всегда FALSE)

    xNfAutoSwitch    : BOOL;   // ← DI11, ручка режима фильтрации = АВТО
    xNfManualSwitch  : BOOL;   // ← DI12, ручка режима фильтрации = РУЧНОЙ
    xNfManualRelayAlarm : BOOL; // авария: ручной режим (DI12), а DI7=0 более 2с (защёлка)
    sNfModeStatus     : WSTRING(30);  // "Авто"/"Ручной"/"?" — текст режима по DI11/DI12

    (* ===== ОПАСНАЯ СИТУАЦИЯ: СУХОЙ ХОД + РУЧНАЯ ФИЛЬТРАЦИЯ ===== *)
    xDangerCondition       : BOOL;   // = xDryRunAlarm AND xNfManualSwitch, живая
    xDangerCondition_Prev  : BOOL;   // для детекта фронта появления
    xShowDangerDialog      : BOOL;   // видимость диалога — привязать к элементу экрана
    xConfirmDangerDialog   : BOOL;   // кнопка "ОК" пишет сюда := TRUE

    (* ===== ВЫХОДЫ-КОМАНДЫ ================================ *)
    xUvCmd    : BOOL;                // 60ЛО: не используется (выхода на УФ нет)
    xPumpsCmd : BOOL;                // → DO2
    xLightCmd : BOOL;                // → DO3

    (* ===== pH — 60ЛО: не используется целиком, дозация на другом контроллере === *)
    xPhEnable    : BOOL;
    xPhRunCmd    : BOOL;
    xPhOutput    : BOOL;
    xPhRelayFb   : BOOL;
    xPhManualRun : BOOL;
    iPhRunMinToday  : INT;
    iPhRunMinBuffer : INT;
    xPhRelayAlarm : BOOL;

    (* ===== АЛЬГИЦИД — 60ЛО: не используется целиком =========== *)
    xAlgEnable    : BOOL;
    xAlgRunCmd    : BOOL;
    xAlgOutput    : BOOL;
    iAlgAutoStartCount : INT;
    xAlgRelayFb   : BOOL;
    xAlgManualRun : BOOL;
    iAlgManRunSecAccum  : DINT;
    iAlgManRunHour : INT;
    iAlgManRunMin  : INT;
    iAlgManRunSec   : INT;
    xAlgManualTimeStart : BOOL;
    xAlgManualTimeStop  : BOOL;
    xAlgManualTimeRun   : BOOL;
    xAskAlgManualTimeStart : BOOL;
    iAlgManSetMin    : INT;
    iAlgManRemMinRaw    : INT;
    iAlgManRemSecRaw    : INT;
    iAlgManRemHour   : INT;
    iAlgManRemMin : INT;
    iAlgManRemSec : INT;
    rAlgRemainSec  : REAL;
    iAlgRemainHour : INT;
    iAlgRemainMin  : INT;
    iAlgRemainSec  : INT;
    rAlgNextDoseSec : REAL;
    iAlgNextHour : INT;
    iAlgNextMin  : INT;
    iAlgNextSec  : INT;
    rAlgDoseSecCalc : REAL;
    iAlgDoseHour : INT;
    iAlgDoseMin : INT;
    iAlgDoseSec : INT;
    iAlgRunMin  : INT;
    iAlgRunMinBuffer : INT;
    iAlgStartToday   : INT;
    xAlgAlarm        : BOOL;
    rAlgFlowLPerHour : REAL;
    xAlgDosing           : BOOL;
    sAlgDosingStatus     : WSTRING(10);
    iAlgDebtMin      : INT;
    iAlgDebtSec      : INT;
    iAlgDebtHour     : INT;
    sAlgLastDebtTime : WSTRING(30);
    iAlgLastDoseHour : INT;
    iAlgLastDoseMin  : INT;
    iAlgLastDoseSec  : INT;
    sAlgLastDoseTime : WSTRING(30);
    xAlgRelayAlarm : BOOL;

    (* ===== БИОПАГ — 60ЛО: не используется целиком ============== *)
    xBioRunCmd          : BOOL;
    xBioOutput          : BOOL;
    xBioRelayFb         : BOOL;
    xBioDosing          : BOOL;
    sBioDosingStatus    : WSTRING(10);
    rBioDoseSecCalc     : REAL;
    iBioDoseHour    : INT;
    iBioDoseMin     : INT;
    iBioDoseSec     : INT;
    iBioDebtHour        : INT;
    iBioDebtMin         : INT;
    iBioDebtSec         : INT;
    rBioNextDoseSec     : REAL;
    iBioNextHour    : INT;
    iBioNextMin     : INT;
    iBioNextSec     : INT;
    iBioRunHour : INT;
    iBioRunMin  : INT;
    iBioRunSec   : INT;
    iBioStartToday      : INT;
    iBioDebtDays        : INT;
    iAlgDebtDays        : INT;
    sBioLastDebtTime    : WSTRING(30);
    sBioLastDoseTime    : WSTRING(30);
    iBioLastDoseHour    : INT;
    iBioLastDoseMin     : INT;
    iBioLastDoseSec     : INT;
    xBioAlarm           : BOOL;
    rBioFlowLPerHour    : REAL;
    xBioEnable             : BOOL;
    xBioManualRun          : BOOL;
    iBioManRunSecAccum  : DINT;
    iBioManRunHour : INT;
    iBioManRunMin  : INT;
    iBioManRunSec   : INT;
    xBioManualTimeStart : BOOL;
    xBioManualTimeStop  : BOOL;
    xBioManualTimeRun   : BOOL;
    xAskBioManualTimeStart : BOOL;
    iBioManRemHour    : INT;
    iBioManRemMin : INT;
    iBioManRemSec : INT;
    xBioRelayAlarm : BOOL;

    (* ===== СВЕТ ========================================== *)
    xLightEnable     : BOOL;
    xLightForceOn    : BOOL;          // = "ручной пуск" (iLightSelect=0), OR-приоритет
    xLightFault      : BOOL;          // 60ЛО: не используется, всегда FALSE

    xLightRelayFb    : BOOL;   // ← DI10, подтверждение работы подсветки
    xLightRelayAlarm : BOOL;   // авария: DO3 и DI10 разошлись >2с (защёлка)

    (* ===== РАСЧЁТ ЗАКАТА — диагностика для экрана, АКТИВНО ===== *)
    rSunTimeZone       : REAL;
    iSunsetCorrectMin     : INT;
    xSunsetCorrectEarlier : BOOL;
    xSunsetActive      : BOOL;
    xSunsetCoordError  : BOOL;
    iSunsetHourCalc    : INT;
    iSunsetMinuteCalc  : INT;
    iSunsetTimeLeftH   : INT;
    iSunsetTimeLeftM   : INT;
    iSunsetDayOfYear   : INT;
    xIsWeekend         : BOOL;
    sCurrentDateStr    : WSTRING(12);

    xScheduleLightOut      : BOOL;
    xSchedulePumpOut       : BOOL;
    iScheduleLightOnHour   : INT;
    iScheduleLightOnMinute : INT;
    iScheduleOffHour       : INT;
    iScheduleOffMinute     : INT;
    iSchedulePumpOnHour    : INT;
    iSchedulePumpOnMinute  : INT;

    xLightShowInputFields   : BOOL;
    xLightShowComputedTime  : BOOL;
    xLightShowAlwaysOnText  : BOOL;
    xLightShowAlwaysOffText : BOOL;
    xPumpShowInputFields    : BOOL;
    xPumpShowComputedTime   : BOOL;
    xPumpShowAlwaysOnText   : BOOL;
    xPumpShowAlwaysOffText  : BOOL;
    xOffTimeVisible         : BOOL;

    xLightOuterForcedOn  : BOOL;
    xLightOuterForcedOff : BOOL;
    xPumpOuterForcedOn   : BOOL;
    xPumpOuterForcedOff  : BOOL;

    (* ===== НАСОСЫ ФОНТАНА ================================ *)
    xManualPermissionNasos : BOOL;
    xPumpsManualOn : BOOL;           // 60ЛО: не используется (устар.)
    xPumpsForceOn  : BOOL;           // = "ручной пуск" (iPumpSelect=0), OR-приоритет

    xPumpRelayFb    : BOOL;   // ← DI9, подтверждение работы насосов
    xPumpRelayAlarm : BOOL;   // авария: DO2 и DI9 разошлись >2с (защёлка)

    (* ===== ЗВУК (FUTURE_SOUND) — 60ЛО: не используется ========= *)
    xSoundOnSchedule : BOOL;
    xSoundOutput     : BOOL;
    xSoundManualOn   : BOOL;

    (* ===== ФИЛЬТРАЦИЯ (мониторинг) — 60ЛО: не используется ===== *)
    (* Старая карта ДДЮТ (DI1/DI2/DI3/DI4/DI5) не совпадает с новой *)
    (* картой 60ЛО — переменные оставлены объявленными, но не      *)
    (* присваиваются нигде в PRG_Fountain.st.                       *)
    xFilter1Drive     : BOOL;
    xFilter2Drive     : BOOL;
    xDriveStart       : BOOL;
    xUvContactor      : BOOL;
    xFilter1Contactor : BOOL;
    xManualFilter     : BOOL;

    (* ===== АВАРИИ ======================================== *)
    xAlarmFountain      : BOOL;      // общая авария
    xAlarmReset         : BOOL;

    (* ===== ФЛАГИ ПОДТВЕРЖДЕНИЯ СБРОСА ==================== *)
    xAskResetPh     : BOOL := FALSE;   // 60ЛО: не используется
    xAskResetAlg    : BOOL := FALSE;   // 60ЛО: не используется
    xAskResetBio    : BOOL := FALSE;   // 60ЛО: не используется
    xAskResetRefill : BOOL := FALSE;   // 60ЛО: не используется
    xAskResetNfFlush : BOOL := FALSE;  // АКТИВНО — диалог "Сбросить счётчик промывок?"
    xAskResetAll    : BOOL := FALSE;   // 60ЛО: не используется
    xAskResetAlarms : BOOL := FALSE;   // АКТИВНО — диалог сброса всех аварий
    xConfirmResetPh  : BOOL := FALSE;  // 60ЛО: не используется
    xConfirmResetAlg : BOOL := FALSE;  // 60ЛО: не используется
    xConfirmResetBio : BOOL := FALSE;  // 60ЛО: не используется
    xConfirmResetAll : BOOL := FALSE;  // 60ЛО: не используется
    xConfirmResetRefill  : BOOL := FALSE;  // 60ЛО: не используется
    xConfirmResetNfFlush : BOOL := FALSE;  // АКТИВНО — реальный ST-код в PRG_Fountain

    (* ===== МИГАНИЕ ====================================== *)
    xBlinkFast : BOOL;
    xBlinkSlow : BOOL;

    (* ===== СТРОКОВЫЕ СТАТУСЫ ============================= *)
    sVseSistStatus    : WSTRING(30);
    sPermissionStatus : WSTRING(30);   // насосы фонтана
    sNfEnableStatus   : WSTRING(30);   // 60ЛО: не используется
    sPhStatus         : WSTRING(30);   // 60ЛО: не используется
    sAlgStatus         : WSTRING(30);  // 60ЛО: не используется
    sBioStatus         : WSTRING(30);  // 60ЛО: не используется
    sLightStatus      : WSTRING(30);
    sSoundStatus      : WSTRING(30);   // 60ЛО: не используется
    sRefillStatus     : WSTRING(30);   // 60ЛО: не используется
    sAlarmStopStatus  : WSTRING(30);
    sAlarmCauses      : WSTRING(255);
    sNfStatus         : WSTRING(30);
    sNfHealthyStatus  : WSTRING(30);

    (* ===== ВРЕМЯ (RTC) ================================== *)
    iCurrentYear         : INT;
    iCurrentMonth        : INT;
    iCurrentDay          : INT;
    iCurrentHour         : INT;
    iCurrentMinute       : INT;
    iCurrentSecond       : INT;
    iCurrentTotalMinutes : INT;

    (* === 60ЛО:УДАЛИТЬ ЦЕЛИКОМ — ПР200 и резерв полива СПК ======= *)
    (* Файлы PRG_PR200.st и PRG_PolivSPK.st выводятся из проекта.  *)
    (* Все переменные ниже нужны были только для их компиляции.     *)
    (*
    wPr200SuhoyHod_Net, wPr200Podpitka_Net, wPr200Norma_Net,
    wPr200Pereliv_Net, wPr200Delay_Net, wPr200LevelRead, wPr200StatusRead,
    rPr200SuhoyHod_Cur, rPr200Podpitka_Cur, rPr200Norma_Cur, rPr200Pereliv_Cur,
    rPr200Delay_Cur, rPr200LevelCm, rPr200SuhoyHod_New, rPr200Podpitka_New,
    rPr200Norma_New, rPr200Pereliv_New, rPr200Delay_New,
    wPr200SuhoyHod_Write, wPr200Podpitka_Write, wPr200Norma_Write,
    wPr200Pereliv_Write, wPr200Delay_Write, wPr200ApplyCmd,
    xPr200Online, xPr200DoborActive, xPr200SlivActive, xPr200PolivActive,
    xPr200ErrDobor, xPr200ErrSliv, xPr200ErrPoliv, xApplyBtn,
    xSpkPolivMode, xSpkRawDI17, xSpkRawDI18, xSpkPolivMode_OLD,
    xPr200OnlineStable, iPr200CommFilterSec, xSpkLevelSensorOk,
    xMsgPr200Offline, xMsgSpkNoSensor, xSpkDI_Dobor, xSpkDI_Poliv,
    xSpkDO_Dobor, xSpkDO_Poliv, xSpkRuchDobor, xSpkRuchPoliv,
    xSpkZapDobor, xSpkZapPoliv, xSpkDoborOn, xSpkPolivOn, xSpkErrDobor,
    xSpkErrPoliv, xSpkErrPereliv, iSpkErrDelaySec, sSpkDoborStatus,
    sSpkPolivStatus, sSpkManualStatus, wSpkMV_Inputs, xSpkMV_Error,
    xSpkDI, wSpkMU_Outputs, wSpkMU_OutputsRead, xSpkMU_Error,
    wSpkMU_SafeOutputs, xSpkMU_WriteSafe, xSpkDO, rSpkLevelRaw, xSpkAI_Error
    *)
END_VAR

(* ---- F_FaultCodeToText.st ---- *)
FUNCTION F_FaultCodeToText : WSTRING(100)
(* Без изменений относительно проекта ДДЮТ *)
VAR_INPUT
    eType    : E_PumpType;
    wCode    : WORD;
END_VAR
VAR
    wCleanCode : WORD;
    iCode      : INT;
END_VAR

CASE eType OF

    E_PumpType.PUMP:
        wCleanCode := wCode AND 16#7FFF;
        iCode := WORD_TO_INT(wCleanCode);

        CASE iCode OF
            0:  F_FaultCodeToText := "Нет ошибок";
            1:  F_FaultCodeToText := "OC0: Перегруз по току в режиме Стоп";
            2:  F_FaultCodeToText := "OC1: Перегруз по току при ускорении";
            3:  F_FaultCodeToText := "OC2: Перегруз по току при замедлении";
            4:  F_FaultCodeToText := "OC3: Перегруз по току в работе";
            5:  F_FaultCodeToText := "OU1: Перенапряжение при ускорении";
            6:  F_FaultCodeToText := "OU2: Перенапряжение при замедлении";
            7:  F_FaultCodeToText := "OU3: Перенапряжение в работе";
            9:  F_FaultCodeToText := "LU: Низкое напряжение питания";
            10: F_FaultCodeToText := "OL2: Перегрузка ПЧ";
            11: F_FaultCodeToText := "OL1: Перегрузка двигателя по току";
            14: F_FaultCodeToText := "OH: Перегрев ПЧ";
            15: F_FaultCodeToText := "EF: Аварийная остановка";
            16: F_FaultCodeToText := "CO: Ошибка коммуникации Modbus";
            20: F_FaultCodeToText := "Обрыв сигнала ОС ПИД";
            24: F_FaultCodeToText := "LP: Нижний уровень аварии ОС ПИД";
            27: F_FaultCodeToText := "HP: Верхний уровень аварии ОС ПИД";
            28: F_FaultCodeToText := "LL: Сухой ход";
            29: F_FaultCodeToText := "tE: Превышено время работы";
            31: F_FaultCodeToText := "Pr: Ошибка записи параметра";
        ELSE
            CASE iCode OF
                64: F_FaultCodeToText := "UC0: Внутр. ошибка в Стоп";
                65: F_FaultCodeToText := "UC1: Внутр. ошибка при ускорении";
                66: F_FaultCodeToText := "UC2: Внутр. ошибка при замедлении";
                67: F_FaultCodeToText := "UC3: Внутр. ошибка в работе";
                68: F_FaultCodeToText := "OC0: Перегруз по току в Стоп";
                69: F_FaultCodeToText := "OC1: Перегруз по току при ускорении";
                70: F_FaultCodeToText := "OC2: Перегруз по току при замедлении";
                71: F_FaultCodeToText := "OC3: Перегруз по току в работе";
                80: F_FaultCodeToText := "OU0: Перенапряжение в Стоп";
                81: F_FaultCodeToText := "OU1: Перенапряжение при ускорении";
                82: F_FaultCodeToText := "OU2: Перенапряжение при замедлении";
                83: F_FaultCodeToText := "OU3: Перенапряжение в работе";
                88: F_FaultCodeToText := "LU0: Низкое напряжение в Стоп";
                89: F_FaultCodeToText := "LU1: Низкое напряжение при ускорении";
                90: F_FaultCodeToText := "LU2: Низкое напряжение при замедлении";
                91: F_FaultCodeToText := "LU3: Низкое напряжение в работе";
                92: F_FaultCodeToText := "OL0: Перегрузка ПЧ в Стоп";
                93: F_FaultCodeToText := "OL1: Перегрузка ПЧ при ускорении";
                94: F_FaultCodeToText := "OL2: Перегрузка ПЧ при замедлении";
                95: F_FaultCodeToText := "OL3: Перегрузка ПЧ в работе";
                96: F_FaultCodeToText := "OT0: Перегрузка двиг. в Стоп";
                97: F_FaultCodeToText := "OT1: Перегрузка двиг. при ускорении";
                98: F_FaultCodeToText := "OT2: Перегрузка двиг. при замедлении";
                99: F_FaultCodeToText := "OT3: Перегрузка двиг. в работе";
                100: F_FaultCodeToText := "OH0: Перегрев ПЧ в Стоп";
                101: F_FaultCodeToText := "OH1: Перегрев ПЧ при ускорении";
                102: F_FaultCodeToText := "OH2: Перегрев ПЧ при замедлении";
                103: F_FaultCodeToText := "OH3: Перегрев ПЧ в работе";
                104: F_FaultCodeToText := "ES: Авар. остановка / обрыв фазы";
            ELSE
                F_FaultCodeToText := WCONCAT("Ошибка PUMP код ", INT_TO_WSTRING(iCode));
            END_CASE;
        END_CASE;

    E_PumpType.MINI:
        iCode := WORD_TO_INT(wCode);
        IF (iCode <= 63) OR ((iCode >= 88) AND (iCode <= 91)) THEN
            F_FaultCodeToText := "Нет ошибок";
        ELSE
            CASE iCode OF
                64: F_FaultCodeToText := "UC0: Внутр. ошибка в Стоп";
                65: F_FaultCodeToText := "UC1: Внутр. ошибка при ускорении";
                66: F_FaultCodeToText := "UC2: Внутр. ошибка при замедлении";
                67: F_FaultCodeToText := "UC3: Внутр. ошибка в работе";
                68: F_FaultCodeToText := "OC0: Перегруз по току в Стоп";
                69: F_FaultCodeToText := "OC1: Перегруз по току при ускорении";
                70: F_FaultCodeToText := "OC2: Перегруз по току при замедлении";
                71: F_FaultCodeToText := "OC3: Перегруз по току в работе";
                80: F_FaultCodeToText := "OU0: Перенапряжение в Стоп";
                81: F_FaultCodeToText := "OU1: Перенапряжение при ускорении";
                82: F_FaultCodeToText := "OU2: Перенапряжение при замедлении";
                83: F_FaultCodeToText := "OU3: Перенапряжение в работе";
                92: F_FaultCodeToText := "OL0: Перегрузка ПЧ в Стоп";
                93: F_FaultCodeToText := "OL1: Перегрузка ПЧ при ускорении";
                94: F_FaultCodeToText := "OL2: Перегрузка ПЧ при замедлении";
                95: F_FaultCodeToText := "OL3: Перегрузка ПЧ в работе";
                96: F_FaultCodeToText := "OT0: Перегрузка двиг. в Стоп";
                97: F_FaultCodeToText := "OT1: Перегрузка двиг. при ускорении";
                98: F_FaultCodeToText := "OT2: Перегрузка двиг. при замедлении";
                99: F_FaultCodeToText := "OT3: Перегрузка двиг. в работе";
                100: F_FaultCodeToText := "OH0: Перегрев ПЧ в Стоп";
                101: F_FaultCodeToText := "OH1: Перегрев ПЧ при ускорении";
                102: F_FaultCodeToText := "OH2: Перегрев ПЧ при замедлении";
                103: F_FaultCodeToText := "OH3: Перегрев ПЧ в работе";
                104: F_FaultCodeToText := "ES: Авар. остановка / обрыв фазы";
            ELSE
                F_FaultCodeToText := WCONCAT("Ошибка MINI код ", INT_TO_WSTRING(iCode));
            END_CASE;
        END_IF;

END_CASE;

(* ---- F_FormatLogDateOnly.st ---- *)
FUNCTION F_FormatLogDateOnly : WSTRING(10)
(* Дата в формате ДД.ММ.ГГГГ, БЕЗ времени — для сжатого журнала     *)
(* изменений параметров фонтана (F_FountainLogWrite). Без изменений *)
(* относительно проекта ДДЮТ.                                        *)
VAR
    sDay   : WSTRING(4);
    sMonth : WSTRING(4);
END_VAR

IF GVL_Fountain.iCurrentDay < 10 THEN
    sDay := WCONCAT("0", INT_TO_WSTRING(GVL_Fountain.iCurrentDay));
ELSE
    sDay := INT_TO_WSTRING(GVL_Fountain.iCurrentDay);
END_IF;

IF GVL_Fountain.iCurrentMonth < 10 THEN
    sMonth := WCONCAT("0", INT_TO_WSTRING(GVL_Fountain.iCurrentMonth));
ELSE
    sMonth := INT_TO_WSTRING(GVL_Fountain.iCurrentMonth);
END_IF;

F_FormatLogDateOnly := WCONCAT(sDay, WCONCAT(".", WCONCAT(sMonth,
    WCONCAT(".", INT_TO_WSTRING(GVL_Fountain.iCurrentYear)))));

(* ---- F_FormatLogTimestamp.st ---- *)
FUNCTION F_FormatLogTimestamp : WSTRING(20)
(* Без изменений относительно проекта ДДЮТ *)
VAR
    sDay, sMon, sYear, sHour, sMin, sSec : WSTRING(4);
END_VAR
IF iCurrentDay < 10 THEN
    sDay := WCONCAT("0", INT_TO_WSTRING(iCurrentDay));
ELSE sDay := INT_TO_WSTRING(iCurrentDay); END_IF;
IF iCurrentMonth < 10 THEN
    sMon := WCONCAT("0", INT_TO_WSTRING(iCurrentMonth));
ELSE sMon := INT_TO_WSTRING(iCurrentMonth); END_IF;
sYear := INT_TO_WSTRING(iCurrentYear MOD 100);
IF (iCurrentYear MOD 100) < 10 THEN
    sYear := WCONCAT("0", sYear);
END_IF;
IF iCurrentHour < 10 THEN
    sHour := WCONCAT("0", INT_TO_WSTRING(iCurrentHour));
ELSE sHour := INT_TO_WSTRING(iCurrentHour); END_IF;
IF iCurrentMinute < 10 THEN
    sMin := WCONCAT("0", INT_TO_WSTRING(iCurrentMinute));
ELSE sMin := INT_TO_WSTRING(iCurrentMinute); END_IF;
IF iCurrentSecond < 10 THEN
    sSec := WCONCAT("0", INT_TO_WSTRING(iCurrentSecond));
ELSE sSec := INT_TO_WSTRING(iCurrentSecond); END_IF;
F_FormatLogTimestamp := WCONCAT(sDay, WCONCAT(".",
    WCONCAT(sMon, WCONCAT(".",
    WCONCAT(sYear, WCONCAT(" ",
    WCONCAT(sHour, WCONCAT(":",
    WCONCAT(sMin, WCONCAT(":", sSec))))))))));

(* ---- F_FountainLogWrite.st ---- *)
FUNCTION F_FountainLogWrite : BOOL
(* Без изменений относительно проекта ДДЮТ. Позиция 1 — ВСЕГДА    *)
(* самая последняя запись. При новой записи всё содержимое          *)
(* сдвигается на 1 позицию вниз (сдвиг ОБЯЗАТЕЛЬНО с конца массива   *)
(* к началу — иначе затрёшь данные раньше, чем скопируешь), новая    *)
(* запись садится на 1. Когда достигнут предел (60) — самая старая   *)
(* запись (позиция 60) просто выпадает при сдвиге. Экран использует  *)
(* ФИКСИРОВАННЫЕ индексы (aFountainLog[1], [2], [3]...).             *)
VAR_INPUT
    sChangeText : WSTRING(60);   (* полное понятное название параметра: старое→новое *)
END_VAR
VAR
    i : INT;
END_VAR

FOR i := 60 TO 2 BY -1 DO
    GVL_Fountain.aFountainLog[i] := GVL_Fountain.aFountainLog[i-1];
END_FOR;

GVL_Fountain.aFountainLog[1] := WCONCAT(F_FormatLogDateOnly(), WCONCAT(" ", sChangeText));

IF GVL_Fountain.iFountainLogCount < 60 THEN
    GVL_Fountain.iFountainLogCount := GVL_Fountain.iFountainLogCount + 1;
END_IF;

F_FountainLogWrite := TRUE;

(* ---- F_LightScheduleModeText.st ---- *)
FUNCTION F_LightScheduleModeText : WSTRING(12)
(* Переводит iLightScheduleMode (0-3) в текст для журнала. ВНИМАНИЕ: *)
(* кодировка ДРУГАЯ, чем у F_SelectModeText — здесь 0=Авто, а не      *)
(* Ручной. Без изменений относительно проекта ДДЮТ.                   *)
VAR_INPUT
    iMode : INT;
END_VAR

CASE iMode OF
    0: F_LightScheduleModeText := "Авто";
    1: F_LightScheduleModeText := "Вкл";
    2: F_LightScheduleModeText := "Выкл";
    3: F_LightScheduleModeText := "Астро";
ELSE
    F_LightScheduleModeText := "?";
END_CASE;

(* ---- F_PumpLogWrite.st ---- *)
FUNCTION F_PumpLogWrite : BOOL
(* Та же схема сдвига, что у F_FountainLogWrite (см. подробный      *)
(* комментарий там) — позиция 1 всегда самая свежая запись, сдвиг    *)
(* ОБЯЗАТЕЛЬНО с конца массива к началу. Без изменений от ДДЮТ.      *)
VAR_INPUT
    sChangeText : WSTRING(65);   (* готовая строка одной записи *)
END_VAR
VAR
    i : INT;
END_VAR

FOR i := 30 TO 2 BY -1 DO
    GVL.aPumpLog[i] := GVL.aPumpLog[i-1];
END_FOR;

GVL.aPumpLog[1] := sChangeText;

IF GVL.iPumpLogCount < 30 THEN
    GVL.iPumpLogCount := GVL.iPumpLogCount + 1;
END_IF;

F_PumpLogWrite := TRUE;

(* ---- F_PumpScheduleModeText.st ---- *)
FUNCTION F_PumpScheduleModeText : WSTRING(12)
(* Переводит iPumpScheduleMode (0-2, БЕЗ "Астро") в текст для        *)
(* журнала. Своя, третья кодировка. Без изменений от ДДЮТ.            *)
VAR_INPUT
    iMode : INT;
END_VAR

CASE iMode OF
    0: F_PumpScheduleModeText := "Авто";
    1: F_PumpScheduleModeText := "Вкл";
    2: F_PumpScheduleModeText := "Выкл";
ELSE
    F_PumpScheduleModeText := "?";
END_CASE;

(* ---- F_SdLogMonthKey.st ---- *)
(* ============================================================ *)
(* F_SdLogMonthKey — РАЗБОР ИМЕНИ ФАЙЛА ЖУРНАЛА → КЛЮЧ МЕСЯЦА   *)
(* ============================================================ *)
(* Принимает ИМЯ ФАЙЛА (не путь!), как его отдаёт FILE.DirList в  *)
(* deDirEntry.sEntry, и префикс журнала. Если имя ТОЧНО совпадает *)
(* с шаблоном "<префикс>MM-YYYY.log" — возвращает ключ месяца:    *)
(*                                                               *)
(*        КЛЮЧ = YYYY * 12 + (MM - 1)                            *)
(*                                                               *)
(* Ключ монотонно растёт со временем, поэтому "самый старый       *)
(* месяц" = минимальный ключ. Декабрь 2025 = 24311, январь 2026 = *)
(* 24312 — переход через год сравнивается правильно, в отличие от *)
(* сравнения строк "12-2025" и "01-2026".                        *)
(*                                                               *)
(* Возвращает 0, если имя НЕ подходит под шаблон. Ноль как признак*)
(* "не наш файл" безопасен: минимально возможный реальный ключ =  *)
(* 2000*12 = 24000, нулём он не станет никогда.                  *)
(*                                                               *)
(* ⚠️ ГЛАВНОЕ НАЗНАЧЕНИЕ — ЗАЩИТА ОТ УДАЛЕНИЯ ЧУЖИХ ФАЙЛОВ.       *)
(* Проверяется ВСЁ: длина имени, префикс, что MM и YYYY — цифры,  *)
(* разделители '-' и '.', расширение 'log', диапазоны MM 1..12 и  *)
(* YYYY 2000..2199. Любое несовпадение → 0 → файл не тронут.      *)
(* Регистр букв игнорируется (FAT может отдать имя иначе).        *)
(* ============================================================ *)
FUNCTION F_SdLogMonthKey : UDINT
VAR_INPUT
    sName   : STRING(255);  (* имя файла из DirList, без пути *)
    sPrefix : STRING(20);   (* 'alarms-' / 'pump_changes-' / 'setpoints-' *)
END_VAR
VAR
    iLenName : INT;
    iLenPref : INT;
    iOfs     : INT;
    i        : INT;
    bN       : BYTE;
    bP       : BYTE;
    iMM      : INT;
    iYY      : INT;
END_VAR

F_SdLogMonthKey := 0;

iLenPref := LEN(sPrefix);
iLenName := LEN(sName);

(* "MM-YYYY.log" — ровно 11 символов после префикса *)
IF iLenPref = 0 OR iLenName <> iLenPref + 11 THEN
    RETURN;
END_IF;

(* --- префикс, без учёта регистра --- *)
FOR i := 0 TO iLenPref - 1 DO
    bN := sName[i];
    bP := sPrefix[i];
    IF bN >= 65 AND bN <= 90 THEN bN := bN + 32; END_IF;   // 'A'..'Z' → нижний
    IF bP >= 65 AND bP <= 90 THEN bP := bP + 32; END_IF;
    IF bN <> bP THEN
        RETURN;
    END_IF;
END_FOR;

iOfs := iLenPref;

(* --- MM (2 цифры) --- *)
iMM := 0;
FOR i := iOfs TO iOfs + 1 DO
    bN := sName[i];
    IF bN < 48 OR bN > 57 THEN RETURN; END_IF;             // не цифра
    iMM := iMM * 10 + BYTE_TO_INT(bN) - 48;
END_FOR;

(* --- разделитель '-' --- *)
IF sName[iOfs + 2] <> 45 THEN RETURN; END_IF;

(* --- YYYY (4 цифры) --- *)
iYY := 0;
FOR i := iOfs + 3 TO iOfs + 6 DO
    bN := sName[i];
    IF bN < 48 OR bN > 57 THEN RETURN; END_IF;
    iYY := iYY * 10 + BYTE_TO_INT(bN) - 48;
END_FOR;

(* --- точка --- *)
IF sName[iOfs + 7] <> 46 THEN RETURN; END_IF;

(* --- расширение 'log' без учёта регистра --- *)
bN := sName[iOfs + 8];
IF bN >= 65 AND bN <= 90 THEN bN := bN + 32; END_IF;
IF bN <> 108 THEN RETURN; END_IF;                          // 'l'
bN := sName[iOfs + 9];
IF bN >= 65 AND bN <= 90 THEN bN := bN + 32; END_IF;
IF bN <> 111 THEN RETURN; END_IF;                          // 'o'
bN := sName[iOfs + 10];
IF bN >= 65 AND bN <= 90 THEN bN := bN + 32; END_IF;
IF bN <> 103 THEN RETURN; END_IF;                          // 'g'

(* --- диапазоны --- *)
IF iMM < 1 OR iMM > 12 THEN RETURN; END_IF;
IF iYY < 2000 OR iYY > 2199 THEN RETURN; END_IF;

F_SdLogMonthKey := INT_TO_UDINT(iYY) * 12 + INT_TO_UDINT(iMM) - 1;

(* ---- F_SdLogPath.st ---- *)
(* ============================================================ *)
(* F_SdLogPath — ПОЛНЫЙ ПУТЬ К ПОМЕСЯЧНОМУ ЖУРНАЛУ НА SD        *)
(* ============================================================ *)
(* Собирает "<каталог>/<префикс>MM-YYYY.log", например:          *)
(*   F_SdLogPath('/mnt/ufs/media/mmcblk0p1', 'alarms-', 2026, 8) *)
(*   → '/mnt/ufs/media/mmcblk0p1/alarms-08-2026.log'             *)
(*                                                               *)
(* ⚠️ Каталог передавать БЕЗ завершающего '/' — слэш добавляется  *)
(* здесь. Месяц дополняется нулём до 2 знаков, год — ВСЕГДА 4     *)
(* знака (вызывающий обязан проверить диапазон 2000..2199, см.    *)
(* PRG_AlarmLogSD блок 4). Ровно 11 символов "MM-YYYY.log" после  *)
(* префикса — на это же число опирается разбор в F_SdLogMonthKey. *)
(*                                                               *)
(* Длина результата: 24 (путь SD) + 1 + 13 (самый длинный         *)
(* префикс 'pump_changes-') + 11 = 49 символов, в STRING(80)      *)
(* помещается с запасом.                                         *)
(* ============================================================ *)
FUNCTION F_SdLogPath : STRING(80)
VAR_INPUT
    sDir    : STRING(80);   (* каталог на карте, БЕЗ '/' в конце *)
    sPrefix : STRING(20);   (* 'alarms-' / 'pump_changes-' / 'setpoints-' *)
    iYear   : INT;          (* 2000..2199 *)
    iMonth  : INT;          (* 1..12 *)
END_VAR
VAR
    sMM : STRING(4);
    sYY : STRING(8);
END_VAR

sMM := INT_TO_STRING(iMonth);
IF iMonth < 10 THEN
    sMM := CONCAT('0', sMM);
END_IF;

sYY := INT_TO_STRING(iYear);

F_SdLogPath := CONCAT(sDir,
               CONCAT('/',
               CONCAT(sPrefix,
               CONCAT(sMM,
               CONCAT('-',
               CONCAT(sYY, '.log'))))));

(* ---- F_SelectModeText.st ---- *)
FUNCTION F_SelectModeText : WSTRING(12)
(* Переводит 0/1/2 (единый селектор насосов/света) в читаемый текст  *)
(* для журнала изменений. Без изменений относительно проекта ДДЮТ.    *)
VAR_INPUT
    iMode : INT;
END_VAR

CASE iMode OF
    0: F_SelectModeText := "Ручной";
    1: F_SelectModeText := "Выкл";
    2: F_SelectModeText := "Авто";
ELSE
    F_SelectModeText := "?";
END_CASE;

(* ---- FB_FountainSchedule.st ---- *)
(* ================================================================
   FB_FountainSchedule — Расписание Фонтана (свет + насосы)
   Без изменений относительно проекта ДДЮТ.

   СВЕТ (Light_Mode, UDINT, 4 положения):
     0 = АВТО, 1 = ВКЛ, 2 = ВЫКЛ, 3 = АСТРО

   НАСОСЫ (Pump_Mode, UDINT, 3 положения — БЕЗ режима "Астро"):
     0 = АВТО, 1 = ВКЛ, 2 = ВЫКЛ

   ВАЖНО: это ВНУТРЕННИЙ выбор — работает только когда ВНЕШНИЙ
   селектор узла (GVL_Fountain.iLightSelect / iPumpSelect) стоит
   в положении "Авто" (=2).
   ================================================================ *)

FUNCTION_BLOCK FB_FountainSchedule

VAR_INPUT
    Sunset_Auto         : BOOL;
    Sunset_Hour         : UDINT;
    Sunset_Minute       : UDINT;
    IsWeekend           : BOOL;

    Light_Mode          : UDINT;

    Light_On_Hour_Weekday   : UDINT;
    Light_On_Minute_Weekday : UDINT;
    Light_On_Hour_Weekend   : UDINT;
    Light_On_Minute_Weekend : UDINT;

    Off_Hour_Weekday    : UDINT;
    Off_Minute_Weekday  : UDINT;
    Off_Hour_Weekend    : UDINT;
    Off_Minute_Weekend  : UDINT;

    Pump_Mode                : UDINT;

    Pump_On_Hour_Weekday    : UDINT;
    Pump_On_Minute_Weekday  : UDINT;
    Pump_On_Hour_Weekend    : UDINT;
    Pump_On_Minute_Weekend  : UDINT;

    Sys_Hour            : UDINT;
    Sys_Minute          : UDINT;
END_VAR

VAR_OUTPUT
    Light_Out             : BOOL;
    Pump_Out               : BOOL;

    Light_On_Result_Hour   : UDINT;
    Light_On_Result_Minute : UDINT;

    Pump_On_Result_Hour     : UDINT;
    Pump_On_Result_Minute   : UDINT;

    Off_Result_Hour         : UDINT;
    Off_Result_Minute       : UDINT;

    Light_ShowInputFields    : BOOL;
    Light_ShowComputedTime   : BOOL;
    Light_ShowAlwaysOnText   : BOOL;
    Light_ShowAlwaysOffText  : BOOL;

    Pump_ShowInputFields     : BOOL;
    Pump_ShowComputedTime    : BOOL;
    Pump_ShowAlwaysOnText    : BOOL;
    Pump_ShowAlwaysOffText   : BOOL;

    Off_Time_Visible          : BOOL;
END_VAR

VAR
    now_total_min       : UDINT;
    light_on_min         : UDINT;
    light_off_min        : UDINT;
    pump_on_min           : UDINT;
    pump_off_min          : UDINT;
    off_today_min         : UDINT;
END_VAR

now_total_min := Sys_Hour * 60 + Sys_Minute;

IF IsWeekend THEN
    off_today_min := Off_Hour_Weekend * 60 + Off_Minute_Weekend;
ELSE
    off_today_min := Off_Hour_Weekday * 60 + Off_Minute_Weekday;
END_IF;

(* ================== СВЕТ ================== *)
IF Light_Mode = 0 THEN
    IF IsWeekend THEN
        light_on_min := Light_On_Hour_Weekend * 60 + Light_On_Minute_Weekend;
    ELSE
        light_on_min := Light_On_Hour_Weekday * 60 + Light_On_Minute_Weekday;
    END_IF;
    light_off_min := off_today_min;

    IF light_off_min > light_on_min THEN
        Light_Out := (now_total_min >= light_on_min) AND (now_total_min < light_off_min);
    ELSE
        Light_Out := (now_total_min >= light_on_min) OR (now_total_min < light_off_min);
    END_IF;

ELSIF Light_Mode = 1 THEN
    Light_Out := TRUE;

ELSIF Light_Mode = 3 THEN
    light_on_min  := Sunset_Hour * 60 + Sunset_Minute;
    light_off_min := off_today_min;

    IF light_off_min > light_on_min THEN
        Light_Out := (now_total_min >= light_on_min) AND (now_total_min < light_off_min);
    ELSE
        Light_Out := (now_total_min >= light_on_min) OR (now_total_min < light_off_min);
    END_IF;

ELSE
    Light_Out := FALSE;
END_IF;

IF Light_Mode = 0 THEN
    IF IsWeekend THEN
        Light_On_Result_Hour   := Light_On_Hour_Weekend;
        Light_On_Result_Minute := Light_On_Minute_Weekend;
    ELSE
        Light_On_Result_Hour   := Light_On_Hour_Weekday;
        Light_On_Result_Minute := Light_On_Minute_Weekday;
    END_IF;
ELSIF Light_Mode = 3 THEN
    Light_On_Result_Hour   := Sunset_Hour;
    Light_On_Result_Minute := Sunset_Minute;
ELSE
    Light_On_Result_Hour   := 0;
    Light_On_Result_Minute := 0;
END_IF;

Light_ShowInputFields   := (Light_Mode = 0);
Light_ShowComputedTime  := (Light_Mode = 0) OR (Light_Mode = 3);
Light_ShowAlwaysOnText  := (Light_Mode = 1);
Light_ShowAlwaysOffText := (Light_Mode = 2);

(* ================== НАСОСЫ ================== *)
IF Pump_Mode = 0 THEN
    IF IsWeekend THEN
        pump_on_min := Pump_On_Hour_Weekend * 60 + Pump_On_Minute_Weekend;
    ELSE
        pump_on_min := Pump_On_Hour_Weekday * 60 + Pump_On_Minute_Weekday;
    END_IF;
    pump_off_min := off_today_min;

    IF pump_off_min > pump_on_min THEN
        Pump_Out := (now_total_min >= pump_on_min) AND (now_total_min < pump_off_min);
    ELSE
        Pump_Out := (now_total_min >= pump_on_min) OR (now_total_min < pump_off_min);
    END_IF;

ELSIF Pump_Mode = 1 THEN
    Pump_Out := TRUE;

ELSE
    Pump_Out := FALSE;
END_IF;

IF Pump_Mode = 0 THEN
    IF IsWeekend THEN
        Pump_On_Result_Hour   := Pump_On_Hour_Weekend;
        Pump_On_Result_Minute := Pump_On_Minute_Weekend;
    ELSE
        Pump_On_Result_Hour   := Pump_On_Hour_Weekday;
        Pump_On_Result_Minute := Pump_On_Minute_Weekday;
    END_IF;
ELSE
    Pump_On_Result_Hour   := 0;
    Pump_On_Result_Minute := 0;
END_IF;

Pump_ShowInputFields   := (Pump_Mode = 0);
Pump_ShowComputedTime  := (Pump_Mode = 0);
Pump_ShowAlwaysOnText  := (Pump_Mode = 1);
Pump_ShowAlwaysOffText := (Pump_Mode = 2);

Off_Result_Hour   := off_today_min / 60;
Off_Result_Minute := off_today_min MOD 60;

Off_Time_Visible := Light_ShowComputedTime OR Pump_ShowComputedTime;

(* ---- FB_Pump.st ---- *)
(* ============================================================ *)
(* FB_Pump — управление одним ПЧ ELHART (PUMP/MINI) по Modbus  *)
(* Без изменений относительно проекта ДДЮТ. Температура (блок 6) *)
(* — без деления на 10 (регистр 0x0006 отдаёт целые °C).          *)
(* ============================================================ *)

FUNCTION_BLOCK FB_Pump
VAR_INPUT
    eType      : E_PumpType;
    xDebugMode : BOOL;
    xCommError : BOOL;
    xCommUnstable : BOOL;

    xRunCmd      : BOOL;
    rFreqSetHz   : REAL;

    wStatus          : WORD;
    wFaultReg        : WORD;
    wFreqSetRead     : WORD;
    wFreqActual      : WORD;
    wCurrentActual   : WORD;
    wSpeedActual     : WORD;
    wDcVoltage       : WORD;
    wTemperature     : WORD;
    wVoltageActual   : WORD;
    wRuntimeHoursRaw : WORD;
    wAccTimeRawRead        : WORD;
    wDecTimeRawRead        : WORD;
    wMaxFreqRead           : WORD;
    wMinFreqRead           : WORD;
    wMotorRatedCurrentRead : WORD;
    wMotorRatedVoltageRead : WORD;
    wOverCurrentLevelRead  : WORD;
    wOverheatLevelRead     : WORD;
    wOverCurAccRead        : WORD;
    wOverCurrentTimeRead   : WORD;
    wOverVoltProtectRead   : WORD;

    rAccTime_Set            : REAL;
    rDecTime_Set            : REAL;
    rMaxFreq_Set            : REAL;
    rMinFreq_Set            : REAL;
    rMotorRatedCurrent_Set  : REAL;
    rMotorRatedVoltage_Set  : REAL;
    rOverCurrentLevel_A_Set : REAL;
    rOverCurrentTime_Set    : REAL;
    xOverVoltProtect_Set    : BOOL;
    iOverheatLevel_Set      : INT;
    iOverCurAcc_Set         : INT;
END_VAR
VAR_OUTPUT
    wCmd  : WORD;
    wFreq : WORD;
    wAccTimeRawWrite        : WORD;
    wDecTimeRawWrite        : WORD;
    wMaxFreqWrite           : WORD;
    wMinFreqWrite           : WORD;
    wMotorRatedCurrentWrite : WORD;
    wMotorRatedVoltageWrite : WORD;
    wOverCurrentLevelWrite  : WORD;
    wOverCurrentTimeWrite   : WORD;
    wOverVoltProtectWrite   : WORD;
    wOverheatLevelWrite     : WORD;
    wOverCurAccWrite        : WORD;

    xRun       : BOOL;
    xStop      : BOOL;
    xAlarm     : BOOL;
    sState     : WSTRING(50);
    sFaultText : WSTRING(100);
    sTypeText  : WSTRING(20);
    xReverse   : BOOL;

    rFreqSetActHz : REAL;
    rFreqActHz    : REAL;
    rCurrentActA  : REAL;
    rSpeedActRpm  : REAL;
    rDcVoltageV   : REAL;
    iTemperatureC : INT;
    rVoltageActV  : REAL;
    rRuntimeHours : REAL;
    rAccTime_Disp            : REAL;
    rDecTime_Disp            : REAL;
    rMaxFreq_Disp            : REAL;
    rMinFreq_Disp            : REAL;
    rMotorRatedCurrent_Disp  : REAL;
    rMotorRatedVoltage_Disp  : REAL;
    rOverCurrentLevel_A_Disp : REAL;
    iOverCurrentLevel_pct_Disp : INT;
    iOverheatLevel_Disp      : INT;
    iOverCurAcc_Disp         : INT;
    rOverCurrentTime_Disp    : REAL;
    xOverVoltProtect_Disp    : BOOL;
END_VAR
VAR
    rK_Freq         : REAL;
    rFreqLim        : REAL;
    xFaultActive    : BOOL;
    wCleanFaultCode : WORD;
    iFaultCode      : INT;
    rTmp : REAL;
    iTmp : INT;
END_VAR

IF eType = E_PumpType.PUMP THEN
    rK_Freq   := 100.0;
    sTypeText := "EMD-PUMP";
ELSE
    rK_Freq   := 10.0;
    sTypeText := "EMD-MINI v2.1";
END_IF;

rFreqLim := rFreqSetHz;
IF rFreqLim < cMinFreq THEN rFreqLim := cMinFreq; END_IF;
IF rFreqLim > cMaxFreq THEN rFreqLim := cMaxFreq; END_IF;

IF xRunCmd THEN
    wCmd  := 16#000A;
    wFreq := REAL_TO_WORD(rFreqLim * rK_Freq);
ELSE
    wCmd  := 16#0009;
    wFreq := REAL_TO_WORD(rFreqLim * rK_Freq);
END_IF;

xStop := FALSE; xRun := FALSE; xAlarm := FALSE;
xReverse := FALSE; xFaultActive := FALSE;

IF xCommError OR xCommUnstable THEN
    xAlarm     := FALSE;
    xStop      := FALSE;
    xRun       := FALSE;
    sState     := "Нет связи с ПЧ";
    sFaultText := "Проверьте RS-485 / адрес / питание ПЧ";
    RETURN;
END_IF;

CASE eType OF
    E_PumpType.PUMP:
        xReverse := (wStatus AND 16#0004) <> 0;
        IF (wStatus AND 16#0008) <> 0 THEN
            xAlarm := TRUE; xFaultActive := TRUE; sState := "Авария";
        ELSIF (wStatus AND 16#0001) <> 0 THEN
            xRun := TRUE;
            IF xReverse THEN sState := "Работа (реверс)"; ELSE sState := "Работа"; END_IF;
        ELSE
            xStop := TRUE; sState := "Стоп";
        END_IF;
    E_PumpType.MINI:
        xReverse := (wStatus AND 16#0001) <> 0;
        IF (wStatus AND 16#0002) <> 0 THEN
            xRun := TRUE;
            IF xReverse THEN sState := "Работа (реверс)"; ELSE sState := "Работа"; END_IF;
        ELSE
            xStop := TRUE; sState := "Стоп";
        END_IF;
END_CASE;

CASE eType OF
    E_PumpType.PUMP:
        IF (wFaultReg AND 16#8000) <> 0 THEN
            xAlarm := TRUE; xRun := FALSE; xStop := FALSE; sState := "Авария";
            wCleanFaultCode := wFaultReg AND 16#7FFF;
            sFaultText := F_FaultCodeToText(eType, wCleanFaultCode);
        ELSE
            sFaultText := "Нет ошибок";
        END_IF;
    E_PumpType.MINI:
        iFaultCode := WORD_TO_INT(wFaultReg);
        IF (iFaultCode > 63) AND ((iFaultCode < 88) OR (iFaultCode > 91)) THEN
            xAlarm := TRUE; xRun := FALSE; xStop := FALSE; sState := "Авария";
            sFaultText := F_FaultCodeToText(eType, wFaultReg);
        ELSE
            sFaultText := "Нет ошибок";
        END_IF;
END_CASE;

rFreqSetActHz := WORD_TO_REAL(wFreqSetRead) / rK_Freq;
rFreqActHz    := WORD_TO_REAL(wFreqActual)  / rK_Freq;
rCurrentActA  := WORD_TO_REAL(wCurrentActual) / 10.0;
rSpeedActRpm  := WORD_TO_REAL(wSpeedActual);
rDcVoltageV   := WORD_TO_REAL(wDcVoltage) / 10.0;

iTemperatureC := WORD_TO_INT(wTemperature);

rVoltageActV  := WORD_TO_REAL(wVoltageActual) / 10.0;
rRuntimeHours := WORD_TO_REAL(wRuntimeHoursRaw);

rAccTime_Disp           := WORD_TO_REAL(wAccTimeRawRead) / 10.0;
rDecTime_Disp           := WORD_TO_REAL(wDecTimeRawRead) / 10.0;
rMaxFreq_Disp           := WORD_TO_REAL(wMaxFreqRead) / rK_Freq;
rMinFreq_Disp           := WORD_TO_REAL(wMinFreqRead) / rK_Freq;
rMotorRatedCurrent_Disp := WORD_TO_REAL(wMotorRatedCurrentRead) / 10.0;
rMotorRatedVoltage_Disp := WORD_TO_REAL(wMotorRatedVoltageRead) / 10.0;
iOverCurrentLevel_pct_Disp := WORD_TO_INT(wOverCurrentLevelRead);
IF rMotorRatedCurrent_Disp > 0.0 THEN
    rOverCurrentLevel_A_Disp := (INT_TO_REAL(iOverCurrentLevel_pct_Disp) / 100.0)
                                 * rMotorRatedCurrent_Disp;
ELSE
    rOverCurrentLevel_A_Disp := 0.0;
END_IF;
iOverheatLevel_Disp := WORD_TO_INT(wOverheatLevelRead);
iOverCurAcc_Disp    := WORD_TO_INT(wOverCurAccRead);
rOverCurrentTime_Disp := WORD_TO_REAL(wOverCurrentTimeRead) / 10.0;
xOverVoltProtect_Disp := (wOverVoltProtectRead <> WORD#0);

rTmp := rAccTime_Set;
IF rTmp < cMinTime THEN rTmp := cMinTime; ELSIF rTmp > cMaxTime THEN rTmp := cMaxTime; END_IF;
wAccTimeRawWrite := REAL_TO_WORD(rTmp * 10.0);

rTmp := rDecTime_Set;
IF rTmp < cMinTime THEN rTmp := cMinTime; ELSIF rTmp > cMaxTime THEN rTmp := cMaxTime; END_IF;
wDecTimeRawWrite := REAL_TO_WORD(rTmp * 10.0);

rTmp := rMaxFreq_Set;
IF rTmp < 1.0 THEN rTmp := 1.0; ELSIF rTmp > cMaxFreq THEN rTmp := cMaxFreq; END_IF;
wMaxFreqWrite := REAL_TO_WORD(rTmp * rK_Freq);
rTmp := rMinFreq_Set;
IF rTmp < 0.0 THEN rTmp := 0.0; ELSIF rTmp > rMaxFreq_Set THEN rTmp := rMaxFreq_Set; END_IF;
wMinFreqWrite := REAL_TO_WORD(rTmp * rK_Freq);

rTmp := rMotorRatedVoltage_Set;
IF rTmp < 0.0 THEN rTmp := 0.0; ELSIF rTmp > cMaxVoltage THEN rTmp := cMaxVoltage; END_IF;
wMotorRatedVoltageWrite := REAL_TO_WORD(rTmp * 10.0);
rTmp := rMotorRatedCurrent_Set;
IF rTmp < 0.1 THEN rTmp := 0.1; ELSIF rTmp > cMaxCurrent THEN rTmp := cMaxCurrent; END_IF;
wMotorRatedCurrentWrite := REAL_TO_WORD(rTmp * 10.0);

IF rMotorRatedCurrent_Set > 0.0 THEN
    iTmp := REAL_TO_INT((rOverCurrentLevel_A_Set / rMotorRatedCurrent_Set) * 100.0);
ELSE
    iTmp := 0;
END_IF;
IF iTmp < 0 THEN iTmp := 0; ELSIF iTmp > 200 THEN iTmp := 200; END_IF;
wOverCurrentLevelWrite := INT_TO_WORD(iTmp);

rTmp := rOverCurrentTime_Set;
IF rTmp < 0.0 THEN rTmp := 0.0; END_IF;
CASE eType OF
    E_PumpType.PUMP: IF rTmp > 999.9 THEN rTmp := 999.9; END_IF;
    E_PumpType.MINI: IF rTmp > 5.0 THEN rTmp := 5.0; END_IF;
END_CASE;
wOverCurrentTimeWrite := REAL_TO_WORD(rTmp * 10.0);

IF xOverVoltProtect_Set THEN wOverVoltProtectWrite := 1; ELSE wOverVoltProtectWrite := 0; END_IF;

iTmp := iOverheatLevel_Set;
IF iTmp < cMinOverheat THEN iTmp := cMinOverheat; ELSIF iTmp > cMaxOverheat THEN iTmp := cMaxOverheat; END_IF;
wOverheatLevelWrite := INT_TO_WORD(iTmp);

iTmp := iOverCurAcc_Set;
IF iTmp < 0 THEN iTmp := 0; ELSIF iTmp > 200 THEN iTmp := 200; END_IF;
wOverCurAccWrite := INT_TO_WORD(iTmp);

(* ---- FB_SdCardSize.st ---- *)
(* ============================================================ *)
(* FB_SdCardSize — АВТООПРЕДЕЛЕНИЕ ЁМКОСТИ ВСТАВЛЕННОЙ SD        *)
(* ============================================================ *)
(* Читает размер раздела прямо у ядра Linux — ОБЫЧНЫМ ЧТЕНИЕМ    *)
(* ФАЙЛА через CAA File. Никаких дополнительных библиотек, ничего *)
(* не надо разрешать в CODESYSControl.cfg, задача не блокируется. *)
(*                                                               *)
(*   /sys/block/mmcblk0/mmcblk0p1/size                            *)
(*                                                               *)
(* Этот псевдофайл содержит одно число ASCII — количество         *)
(* 512-байтных секторов раздела, например "31116288\n". Отсюда:   *)
(*                                                               *)
(*   ёмкость, МиБ = секторы / 2048     (512 Б * 2048 = 1 МиБ)     *)
(*                                                               *)
(* Дальше вычитаем 1 % на служебные структуры FAT32 (зарезерви-   *)
(* рованные секторы, две копии таблицы FAT, корневой каталог).    *)
(* Для 32 ГБ это ~300 МБ — с запасом, но нам важнее не завысить.  *)
(*                                                               *)
(* ⚠️ ОСОБЕННОСТЬ sysfs: такие файлы часто отдают размер 0, потому *)
(* FILE.GetSize по ним звать нельзя — читаем сразу в буфер на 32  *)
(* байта и смотрим, сколько байт реально пришло (FILE.Read.szSize).*)
(*                                                               *)
(* ⚠️ ЕСЛИ НЕ ПОЛУЧИЛОСЬ (файла нет, другое имя устройства, права) *)
(* — xValid остаётся FALSE, и PRG_AlarmLogSD берёт ёмкость из     *)
(* выпадающего списка на экране. То есть хуже, чем было, не будет  *)
(* никогда: автоопределение — это только удобство.                *)
(*                                                               *)
(* ⚠️ ИМЯ УСТРОЙСТВА. Путь берётся из GVL_Fountain.sSdCardSysPath. *)
(* На СПК карта монтируется в /mnt/ufs/media/mmcblk0p1, поэтому   *)
(* устройство — mmcblk0, раздел — mmcblk0p1. Если на конкретном   *)
(* контроллере SD окажется вторым устройством (mmcblk1p1) —       *)
(* поправить строку в GVL, перекомпиляция логики не нужна.        *)
(* Проверить на месте можно так: значение udiSectors * 512 должно  *)
(* примерно совпасть с объёмом карты.                             *)
(* ============================================================ *)
FUNCTION_BLOCK FB_SdCardSize
VAR_INPUT
    xTrigger : BOOL;          (* ФРОНТ — перечитать размер *)
    sSysPath : STRING(120);   (* '/sys/block/mmcblk0/mmcblk0p1/size' *)
END_VAR
VAR_OUTPUT
    xBusy         : BOOL;
    xValid        : BOOL;     (* ёмкость определена, можно доверять *)
    udiCapacityMB : UDINT;    (* полезная ёмкость, МиБ *)
    udiSectors    : UDINT;    (* сырое значение из sysfs, секторов по 512 Б *)
END_VAR
VAR CONSTANT
    (* разумные границы: меньше 64 МБ и больше 2 ТБ — точно мусор *)
    cMinMB : UDINT := 64;
    cMaxMB : UDINT := 2097152;
END_VAR
VAR
    iSt       : INT;
    xTrigPrev : BOOL;

    fbOpen  : FILE.Open;
    fbRead  : FILE.Read;
    fbClose : FILE.Close;
    hFile   : FILE.CAA.HANDLE;

    abBuf   : ARRAY[0..31] OF BYTE;
    udiRead : UDINT;

    i       : INT;
    b       : BYTE;
    udiSec  : UDINT;
    udiMB   : UDINT;
    iDigits : INT;
END_VAR

(* --- запуск по фронту --- *)
IF xTrigger AND NOT xTrigPrev AND iSt = 0 THEN
    iSt := 1;
END_IF;
xTrigPrev := xTrigger;

xBusy := (iSt <> 0);

CASE iSt OF

    0:  (* IDLE *)
        ;

    1:  (* OPEN на чтение *)
        fbOpen(xExecute := TRUE, sFileName := sSysPath, eFileMode := FILE.MODE.MREAD);
        IF fbOpen.xDone THEN
            hFile := fbOpen.hFile;
            fbOpen(xExecute := FALSE);
            iSt := 2;
        ELSIF fbOpen.xError THEN
            (* нет такого файла / нет доступа — молча уходим на список *)
            fbOpen(xExecute := FALSE);
            xValid := FALSE;
            iSt := 0;
        END_IF;

    2:  (* READ — sysfs отдаёт короткую ASCII-строку *)
        fbRead(xExecute := TRUE, hFile := hFile,
               pBuffer := ADR(abBuf), szBuffer := SIZEOF(abBuf));
        IF fbRead.xDone THEN
            udiRead := fbRead.szSize;
            fbRead(xExecute := FALSE);
            iSt := 3;
        ELSIF fbRead.xError THEN
            fbRead(xExecute := FALSE);
            udiRead := 0;
            iSt := 3;
        END_IF;

    3:  (* CLOSE — закрыть надо в любом случае *)
        fbClose(xExecute := TRUE, hFile := hFile);
        IF fbClose.xDone OR fbClose.xError THEN
            fbClose(xExecute := FALSE);
            iSt := 4;
        END_IF;

    4:  (* РАЗБОР ЧИСЛА *)
        udiSec  := 0;
        iDigits := 0;

        IF udiRead > SIZEOF(abBuf) THEN
            udiRead := SIZEOF(abBuf);
        END_IF;

        FOR i := 0 TO UDINT_TO_INT(udiRead) - 1 DO
            b := abBuf[i];
            IF b >= 48 AND b <= 57 THEN
                (* защита от переполнения UDINT: 429 496 728 * 10 + 9 *)
                (* ещё влезает, больше — уже нет                       *)
                IF udiSec <= 429496728 THEN
                    udiSec  := udiSec * 10 + BYTE_TO_UDINT(b) - 48;
                    iDigits := iDigits + 1;
                ELSE
                    iDigits := 0;      (* число неправдоподобно велико *)
                    EXIT;
                END_IF;
            ELSE
                EXIT;                  (* первый нецифровой символ = конец *)
            END_IF;
        END_FOR;

        IF iDigits > 0 AND udiSec > 0 THEN
            udiSectors := udiSec;
            (* секторы по 512 Б → МиБ, затем −1 % на структуры FAT32 *)
            udiMB := (udiSec / 2048) * 99 / 100;
            IF udiMB >= cMinMB AND udiMB <= cMaxMB THEN
                udiCapacityMB := udiMB;
                xValid := TRUE;
            ELSE
                xValid := FALSE;
            END_IF;
        ELSE
            xValid := FALSE;
        END_IF;

        iSt := 0;

END_CASE;

(* ---- FB_SunsetRelay.st ---- *)
(* ============================================================
   FB_SunsetRelay — Астрономическое реле (расчёт заката)
   Без изменений относительно проекта ДДЮТ.
   Логика:
   - Расчёт времени заката по долготе/широте/часовому поясу
   - Ручная коррекция ±минут (местность: море/горы/рельеф)
   - Выход «Sunset_Auto» = TRUE от заката до времени отключения
   - Точность расчёта: ±1-3 минуты (алгоритм NOAA/Spencer с поправкой
     на атмосферную рефракцию и радиус диска Солнца, угол зенита
     90.833°).
   - Определение будни/выходной (алгоритм Зеллера) — для выбора
     своей пары Off_Hour/Off_Minute, а также выдаётся наружу
     (IsWeekend) для использования в FB_FountainSchedule.
   - Доп. выход: сколько осталось до следующей смены состояния

   ВАЖНО: Sunset_Auto — это ТОЛЬКО автоматический расчёт по закату.
   Финальное управление светом (авто/ручной режим) находится в
   отдельном блоке FB_FountainSchedule — туда подаётся Sunset_Auto
   как один из входов.
   ============================================================ *)

FUNCTION_BLOCK FB_SunsetRelay

VAR_INPUT
    (* --- Геокоординаты с экрана --- *)
    Latitude        : REAL;   (* Широта, градусы  *)
    Longitude       : REAL;   (* Долгота, градусы *)
    TimeZone        : REAL;   (* Часовой пояс, знаковый! ← выход FB_TimeZoneSelect *)

    (* --- Коррекция заката --- *)
    Sunset_Correct  : UDINT;  (* Ручная коррекция заката, минут (0..60)  *)
    Sunset_Earlier   : BOOL;  (* Направление: TRUE = раньше, FALSE = позже *)

    (* --- Настройки отключения: раздельно будни/выходные --- *)
    Off_Hour_Weekday   : UDINT;
    Off_Minute_Weekday : UDINT;
    Off_Hour_Weekend   : UDINT;
    Off_Minute_Weekend : UDINT;

    (* --- Системное время --- *)
    Sys_Year        : UDINT;
    Sys_Month       : UDINT;
    Sys_Day         : UDINT;
    Sys_Hour        : UDINT;
    Sys_Minute      : UDINT;
    Sys_Sec         : UDINT;
END_VAR

VAR_OUTPUT
    Sunset_Auto     : BOOL;   (* Автоматический расчёт: 1 = должно гореть *)
    Sunset_Hour     : UDINT;
    Sunset_Minute   : UDINT;
    DayOfYear       : UDINT;
    Err_Coord       : BOOL;
    IsWeekend       : BOOL;

    Time_Left_H     : UDINT;
    Time_Left_M     : UDINT;
END_VAR

VAR
    i               : UDINT;
    doy             : UDINT;
    lat_rad         : REAL;
    gamma           : REAL;
    eqtime          : REAL;
    decl            : REAL;
    ha              : REAL;
    sunset_utc      : REAL;
    sunset_local    : REAL;
    sunset_total_min : UDINT;
    off_total_min   : UDINT;
    now_total_min   : UDINT;
    diff_min        : UDINT;
    pi              : REAL;
    two_pi          : REAL;
    deg_to_rad      : REAL;
    rad_to_deg      : REAL;
    temp_real       : REAL;
    sunset_corr_real : REAL;
    days_in_month   : ARRAY[1..12] OF UDINT;

    zm              : UDINT;
    zy              : UDINT;
    zK              : UDINT;
    zJ              : UDINT;
    zh              : UDINT;
END_VAR

IF Sys_Month < 3 THEN
    zm := Sys_Month + 12;
    zy := Sys_Year - 1;
ELSE
    zm := Sys_Month;
    zy := Sys_Year;
END_IF;

zK := zy MOD 100;
zJ := zy / 100;

zh := (Sys_Day + (13 * (zm + 1)) / 5 + zK + zK / 4 + zJ / 4 + 5 * zJ) MOD 7;

IsWeekend := (zh = 0) OR (zh = 1);   (* 0=суббота, 1=воскресенье *)

IF IsWeekend THEN
    off_total_min := Off_Hour_Weekend * 60 + Off_Minute_Weekend;
ELSE
    off_total_min := Off_Hour_Weekday * 60 + Off_Minute_Weekday;
END_IF;

pi := 3.14159265;
two_pi := 6.2831853;
deg_to_rad := pi / 180.0;
rad_to_deg := 180.0 / pi;

days_in_month[1] := 31;
days_in_month[2] := 28;
days_in_month[3] := 31;
days_in_month[4] := 30;
days_in_month[5] := 31;
days_in_month[6] := 30;
days_in_month[7] := 31;
days_in_month[8] := 31;
days_in_month[9] := 30;
days_in_month[10] := 31;
days_in_month[11] := 30;
days_in_month[12] := 31;

Err_Coord := (Latitude < -90.0) OR (Latitude > 90.0)
          OR (Longitude < -180.0) OR (Longitude > 180.0);

IF Err_Coord THEN
    Sunset_Auto := FALSE;
    Sunset_Hour := 0;
    Sunset_Minute := 0;
    DayOfYear := 0;
    Time_Left_H := 0;
    Time_Left_M := 0;

ELSE
    doy := 0;
    FOR i := 1 TO 12 DO
        IF i < Sys_Month THEN
            doy := doy + days_in_month[i];
        END_IF;
    END_FOR;
    doy := doy + Sys_Day;

    IF (Sys_Year MOD 4 = 0) THEN
        IF (Sys_Year MOD 100 <> 0) OR (Sys_Year MOD 400 = 0) THEN
            IF Sys_Month > 2 THEN
                doy := doy + 1;
            END_IF;
        END_IF;
    END_IF;
    DayOfYear := doy;

    gamma := two_pi * UDINT_TO_REAL(doy - 1) / 365.0;

    eqtime := 229.18 * (0.000075
             + 0.001868 * COS(gamma)
             - 0.032077 * SIN(gamma)
             - 0.014615 * COS(2.0 * gamma)
             - 0.040849 * SIN(2.0 * gamma));

    decl := 0.006918
          - 0.399912 * COS(gamma)
          + 0.070257 * SIN(gamma)
          - 0.006758 * COS(2.0 * gamma)
          + 0.000907 * SIN(2.0 * gamma)
          - 0.002697 * COS(3.0 * gamma)
          + 0.00148  * SIN(3.0 * gamma);

    lat_rad := Latitude * deg_to_rad;
    temp_real := COS(90.833 * deg_to_rad) / (COS(lat_rad) * COS(decl))
                 - TAN(lat_rad) * TAN(decl);

    IF temp_real > 1.0 THEN
        ha := 0.0;
    ELSIF temp_real < -1.0 THEN
        ha := pi;
    ELSE
        ha := ACOS(temp_real);
    END_IF;

    sunset_utc := 12.0 + (ha * rad_to_deg / 15.0) - (eqtime / 60.0) - (Longitude / 15.0);

    sunset_local := sunset_utc + TimeZone;
    IF sunset_local < 0.0 THEN
        sunset_local := sunset_local + 24.0;
    END_IF;
    IF sunset_local >= 24.0 THEN
        sunset_local := sunset_local - 24.0;
    END_IF;

    sunset_corr_real := UDINT_TO_REAL(Sunset_Correct) / 60.0;
    IF Sunset_Earlier THEN
        sunset_local := sunset_local - sunset_corr_real;
    ELSE
        sunset_local := sunset_local + sunset_corr_real;
    END_IF;

    IF sunset_local < 0.0 THEN
        sunset_local := sunset_local + 24.0;
    END_IF;
    IF sunset_local >= 24.0 THEN
        sunset_local := sunset_local - 24.0;
    END_IF;

    sunset_total_min := REAL_TO_UDINT(sunset_local * 60.0);
    IF sunset_total_min >= 1440 THEN
        sunset_total_min := sunset_total_min - 1440;
    END_IF;
    Sunset_Hour   := sunset_total_min / 60;
    Sunset_Minute := sunset_total_min MOD 60;

    now_total_min := Sys_Hour * 60 + Sys_Minute;

    IF off_total_min > sunset_total_min THEN
        Sunset_Auto := (now_total_min >= sunset_total_min) AND (now_total_min < off_total_min);
    ELSE
        Sunset_Auto := (now_total_min >= sunset_total_min) OR (now_total_min < off_total_min);
    END_IF;

    IF now_total_min < sunset_total_min THEN
        diff_min := sunset_total_min - now_total_min;
    ELSE
        diff_min := (1440 - now_total_min) + sunset_total_min;
    END_IF;

    Time_Left_H := diff_min / 60;
    Time_Left_M := diff_min MOD 60;

END_IF;

(* ---- FB_TimeZoneSelect.st ---- *)
(* ================================================================
   FB_TimeZoneSelect — Выбор часового пояса комбобоксом
   Без изменений относительно проекта ДДЮТ.

   ChoseTimeZone — индекс 0-23 с экрана (Текстовый список).
   Линейная зависимость: TimeZone = ChoseTimeZone - 11.
   ChoseTimeZone = 14 → TimeZone = +3 (Москва) — ЗНАЧЕНИЕ ПО
   УМОЛЧАНИЮ.

   На экране "Текстовый список", строки:
   0  → "-11 Паго-Паго"          12 → "+1  Берлин"
   1  → "-10 Гонолулу"           13 → "+2  Калининград"
   2  → "-9  Анкоридж"           14 → "+3  Москва"   ← ПО УМОЛЧАНИЮ
   3  → "-8  Лос-Анджелес"       15 → "+4  Самара"
   4  → "-7  Денвер"             16 → "+5  Екатеринбург"
   5  → "-6  Мехико"             17 → "+6  Омск"
   6  → "-5  Нью-Йорк"           18 → "+7  Красноярск"
   7  → "-4  Сантьяго"           19 → "+8  Иркутск"
   8  → "-3  Буэнос-Айрес"       20 → "+9  Якутск"
   9  → "-2  Норонья"            21 → "+10 Владивосток"
   10 → "-1  Азорские о-ва"      22 → "+11 Магадан"
   11 → "0   Лондон"             23 → "+12 Камчатка"
   ================================================================ *)

FUNCTION_BLOCK FB_TimeZoneSelect
VAR_INPUT
    ChoseTimeZone   : UDINT;  (* Индекс выбора, 0-23. По умолчанию 14=Москва *)
END_VAR
VAR_OUTPUT
    TimeZone        : REAL;   (* → вход TimeZone в FB_SunsetRelay             *)
END_VAR
VAR
    idx             : UDINT;
END_VAR

IF ChoseTimeZone > 23 THEN
    idx := 14;
ELSE
    idx := ChoseTimeZone;
END_IF;

TimeZone := UDINT_TO_REAL(idx) - 11.0;

END_FUNCTION_BLOCK

(* ---- PLC_PRG.st ---- *)
(* ============================================================ *)
(* PLC_PRG — главная программа (MainTask)                       *)
(* ============================================================ *)
(* ПР200 и резерв полива СПК на "60 Лет Октября" НЕ ИСПОЛЬЗУЮТСЯ *)
(* вообще — файлы PRG_PR200.st / PRG_PolivSPK.st исключены из     *)
(* проекта (были только в ДДЮТ для другого объекта).              *)
(* ============================================================ *)
PROGRAM PLC_PRG
VAR
END_VAR
PRG_IO();         (* распаковка DI, сборка маски DO *)
PRG_Fountain();   (* автоматика фонтана *)
PRG_Pumps();      (* обработка ПЧ-насосов (COM2, теперь 3 шт.) *)
PRG_Errors();     (* подсчёт общих аварий *)
